LIN {X 0,Y 175.394,Z 402.692,A -85,B 0,C 180,E1 -25528.539,E2 -25528.539} C_VEL
LIN {X 0,Y 177.917,Z 390.914,A -85,B 0,C 180,E1 -25529.64,E2 -25529.64} C_VEL
LIN {X 0,Y 179.581,Z 378.992,A -85,B 0,C 180,E1 -25530.439,E2 -25530.439} C_VEL
LIN {X 0,Y 180.606,Z 365.157,A -85,B 0,C 180,E1 -25531.052,E2 -25531.052} C_VEL
LIN {X 0,Y 176.084,Z 356.031,A -85,B 0,C 180,E1 -25534.195,E2 -25534.195} C_VEL
LIN {X 0,Y 171.449,Z 347.762,A -85,B 0,C 180,E1 -25537.875,E2 -25537.875} C_VEL
LIN {X 0,Y 167.95,Z 342.316,A -85,B 0,C 180,E1 -25541.096,E2 -25541.096} C_VEL
LIN {X 0,Y 166.255,Z 339.586,A -85,B 0,C 180,E1 -25542.893,E2 -25542.893} C_VEL
LIN {X 0,Y 163.938,Z 336.007,A -85,B 0,C 180,E1 -25545.689,E2 -25545.689} C_VEL
LIN {X 0,Y 161.573,Z 332.428,A -85,B 0,C 180,E1 -25549.188,E2 -25549.188} C_VEL
LIN {X 0,Y 160.8,Z 331.442,A -85,B 0,C 180,E1 -25550.526,E2 -25550.526} C_VEL
LIN {X 0,Y 158.685,Z 328.085,A -85,B 0,C 180,E1 -25555.56,E2 -25555.56} C_VEL
LIN {X 0,Y 158.317,Z 327.018,A -85,B 0,C 180,E1 -25557.038,E2 -25557.038} C_VEL
LIN {X 0,Y 157.707,Z 326.481,A -85,B 0,C 180,E1 -25559.999,E2 -25559.999} C_VEL
LIN {X 0,Y 158.2,Z 327.003,A -85,B 0,C 180,E1 -25568.944,E2 -25568.944} C_VEL
LIN {X 0,Y 159.684,Z 330.432,A -85,B 0,C 180,E1 -25573.724,E2 -25573.724} C_VEL
LIN {X 0,Y 160.618,Z 331.804,A -85,B 0,C 180,E1 -25575.659,E2 -25575.659} C_VEL
LIN {X 0,Y 161.933,Z 334.433,A -85,B 0,C 180,E1 -25578.055,E2 -25578.055} C_VEL
LIN {X 0,Y 165.141,Z 341.155,A -85,B 0,C 180,E1 -25582.629,E2 -25582.629} C_VEL
LIN {X 0,Y 167.909,Z 347.295,A -85,B 0,C 180,E1 -25585.802,E2 -25585.802} C_VEL
LIN {X 0,Y 170.429,Z 353.215,A -85,B 0,C 180,E1 -25588.32,E2 -25588.32} C_VEL
LIN {X 0,Y 173.374,Z 360.584,A -85,B 0,C 180,E1 -25590.951,E2 -25590.951} C_VEL
LIN {X 0,Y 176.879,Z 370.457,A -85,B 0,C 180,E1 -25593.798,E2 -25593.798} C_VEL
LIN {X 0,Y 177.593,Z 373.058,A -85,B 0,C 180,E1 -25594.381,E2 -25594.381} C_VEL
LIN {X 0,Y 178.04,Z 394.466,A -85,B 0,C 180,E1 -25596.206,E2 -25596.206} C_VEL
LIN {X 0,Y 176.549,Z 407.501,A -85,B 0,C 180,E1 -25596.734,E2 -25596.734} C_VEL
LIN {X 0,Y 173.815,Z 420.614,A -85,B 0,C 180,E1 -25597.525,E2 -25597.525} C_VEL
LIN {X 0,Y 169.933,Z 433.758,A -85,B 0,C 180,E1 -25598.683,E2 -25598.683} C_VEL
LIN {X 0,Y 165.401,Z 445.411,A -85,B 0,C 180,E1 -25600.108,E2 -25600.108} C_VEL
LIN {X 0,Y 159.65,Z 457.154,A -85,B 0,C 180,E1 -25602.024,E2 -25602.024} C_VEL
LIN {X 0,Y 154.205,Z 466.649,A -85,B 0,C 180,E1 -25604.125,E2 -25604.125} C_VEL
LIN {X 0,Y 148.424,Z 475.35,A -85,B 0,C 180,E1 -25606.639,E2 -25606.639} C_VEL
LIN {X 0,Y 142.089,Z 483.85,A -85,B 0,C 180,E1 -25609.983,E2 -25609.983} C_VEL
LIN {X 0,Y 136.434,Z 490.753,A -85,B 0,C 180,E1 -25613.673,E2 -25613.673} C_VEL
LIN {X 0,Y 131.518,Z 496.334,A -85,B 0,C 180,E1 -25617.698,E2 -25617.698} C_VEL
LIN {X 0,Y 127.701,Z 500.475,A -85,B 0,C 180,E1 -25621.709,E2 -25621.709} C_VEL
LIN {X 0,Y 124.221,Z 504.173,A -85,B 0,C 180,E1 -25626.669,E2 -25626.669} C_VEL
LIN {X 0,Y 121.436,Z 507.281,A -85,B 0,C 180,E1 -25633.179,E2 -25633.179} C_VEL
LIN {X 0,Y 120.473,Z 508.774,A -85,B 0,C 180,E1 -25639.92,E2 -25639.92} C_VEL
LIN {X 0,Y 120.585,Z 508.949,A -85,B 0,C 180,E1 -25643.305,E2 -25643.305} C_VEL
LIN {X 0,Y 121.01,Z 508.736,A -85,B 0,C 180,E1 -25646.669,E2 -25646.669} C_VEL
LIN {X 0,Y 121.498,Z 508.07,A -85,B 0,C 180,E1 -25649.999,E2 -25649.999} C_VEL
LIN {X 0,Y 120.971,Z 506.799,A -85,B 0,C 180,E1 -25653.329,E2 -25653.329} C_VEL
LIN {X 0,Y 120.525,Z 504.589,A -85,B 0,C 180,E1 -25657.567,E2 -25657.567} C_VEL
LIN {X 0,Y 120.742,Z 500.25,A -85,B 0,C 180,E1 -25663.462,E2 -25663.462} C_VEL
LIN {X 0,Y 121.918,Z 495.31,A -85,B 0,C 180,E1 -25668.483,E2 -25668.483} C_VEL
LIN {X 0,Y 123.994,Z 489.089,A -85,B 0,C 180,E1 -25673.374,E2 -25673.374} C_VEL
LIN {X 0,Y 127.247,Z 481.256,A -85,B 0,C 180,E1 -25678.099,E2 -25678.099} C_VEL
LIN {X 0,Y 130.569,Z 473.197,A -85,B 0,C 180,E1 -25681.848,E2 -25681.848} C_VEL
LIN {X 0,Y 131.685,Z 468.98,A -85,B 0,C 180,E1 -25683.603,E2 -25683.603} C_VEL
LIN {X 0,Y 132.139,Z 461.767,A -85,B 0,C 180,E1 -25686.543,E2 -25686.543} C_VEL
LIN {X 0,Y 132.615,Z 454.126,A -85,B 0,C 180,E1 -25689.272,E2 -25689.272} C_VEL
LIN {X 0,Y 133.673,Z 449.2,A -85,B 0,C 180,E1 -25690.61,E2 -25690.61} C_VEL
LIN {X 0,Y 137.177,Z 438.275,A -85,B 0,C 180,E1 -25692.75,E2 -25692.75} C_VEL
LIN {X 0,Y 140.428,Z 426.165,A -85,B 0,C 180,E1 -25694.477,E2 -25694.477} C_VEL
LIN {X 0,Y 142.791,Z 413.232,A -85,B 0,C 180,E1 -25695.841,E2 -25695.841} C_VEL
LIN {X 0,Y 144.369,Z 400.263,A -85,B 0,C 180,E1 -25696.68,E2 -25696.68} C_VEL
LIN {X 0,Y 145.125,Z 387.045,A -85,B 0,C 180,E1 -25697.314,E2 -25697.314} C_VEL
LIN {X 0,Y 144.369,Z 355.275,A -85,B 0,C 180,E1 -25699.747,E2 -25699.747} C_VEL
LIN {X 0,Y 143.902,Z 344.092,A -85,B 0,C 180,E1 -25700.717,E2 -25700.717} C_VEL
LIN {X 0,Y 140.398,Z 334.16,A -85,B 0,C 180,E1 -25702.969,E2 -25702.969} C_VEL
LIN {X 0,Y 135.644,Z 322.943,A -85,B 0,C 180,E1 -25706.209,E2 -25706.209} C_VEL
LIN {X 0,Y 132.185,Z 316.035,A -85,B 0,C 180,E1 -25708.763,E2 -25708.763} C_VEL
LIN {X 0,Y 129.855,Z 311.656,A -85,B 0,C 180,E1 -25710.628,E2 -25710.628} C_VEL
LIN {X 0,Y 127.246,Z 306.989,A -85,B 0,C 180,E1 -25712.893,E2 -25712.893} C_VEL
LIN {X 0,Y 124.677,Z 303.799,A -85,B 0,C 180,E1 -25715.213,E2 -25715.213} C_VEL
LIN {X 0,Y 123.773,Z 302.321,A -85,B 0,C 180,E1 -25716.137,E2 -25716.137} C_VEL
LIN {X 0,Y 121.22,Z 299.89,A -85,B 0,C 180,E1 -25718.756,E2 -25718.756} C_VEL
LIN {X 0,Y 119.684,Z 297.038,A -85,B 0,C 180,E1 -25720.713,E2 -25720.713} C_VEL
LIN {X 0,Y 116.749,Z 294.976,A -85,B 0,C 180,E1 -25724.531,E2 -25724.531} C_VEL
LIN {X 0,Y 115.469,Z 292.543,A -85,B 0,C 180,E1 -25726.875,E2 -25726.875} C_VEL
LIN {X 0,Y 115.306,Z 291.427,A -85,B 0,C 180,E1 -25728.301,E2 -25728.301} C_VEL
LIN {X 0,Y 115.34,Z 291.094,A -85,B 0,C 180,E1 -25733.001,E2 -25733.001} C_VEL
LIN {X 0,Y 115.939,Z 291.002,A -85,B 0,C 180,E1 -25740.001,E2 -25740.001} C_VEL
LIN {X 0,Y 115.336,Z 291.08,A -85,B 0,C 180,E1 -25747.001,E2 -25747.001} C_VEL
LIN {X 0,Y 115.198,Z 291.126,A -85,B 0,C 180,E1 -25752.558,E2 -25752.558} C_VEL
LIN {X 0,Y 114.963,Z 291.274,A -85,B 0,C 180,E1 -25760.114,E2 -25760.114} C_VEL
LIN {X 0,Y 115.129,Z 292.227,A -85,B 0,C 180,E1 -25762.246,E2 -25762.246} C_VEL
LIN {X 0,Y 116.662,Z 295.146,A -85,B 0,C 180,E1 -25765.179,E2 -25765.179} C_VEL
LIN {X 0,Y 119.689,Z 297.275,A -85,B 0,C 180,E1 -25769.122,E2 -25769.122} C_VEL
LIN {X 0,Y 121.495,Z 300.418,A -85,B 0,C 180,E1 -25771.375,E2 -25771.375} C_VEL
LIN {X 0,Y 124.006,Z 302.79,A -85,B 0,C 180,E1 -25773.911,E2 -25773.911} C_VEL
LIN {X 0,Y 126.412,Z 306.25,A -85,B 0,C 180,E1 -25776.208,E2 -25776.208} C_VEL
LIN {X 0,Y 127.814,Z 307.903,A -85,B 0,C 180,E1 -25777.405,E2 -25777.405} C_VEL
LIN {X 0,Y 131.403,Z 312.946,A -85,B 0,C 180,E1 -25780.275,E2 -25780.275} C_VEL
LIN {X 0,Y 136.614,Z 320.749,A -85,B 0,C 180,E1 -25783.917,E2 -25783.917} C_VEL
LIN {X 0,Y 141.926,Z 329.84,A -85,B 0,C 180,E1 -25787.192,E2 -25787.192} C_VEL
LIN {X 0,Y 147.468,Z 341.166,A -85,B 0,C 180,E1 -25790.295,E2 -25790.295} C_VEL
LIN {X 0,Y 148.103,Z 342.665,A -85,B 0,C 180,E1 -25790.639,E2 -25790.639} C_VEL
LIN {X 0,Y 145.968,Z 378.464,A -85,B 0,C 180,E1 -25792.341,E2 -25792.341} C_VEL
LIN {X 0,Y 144.546,Z 391.684,A -85,B 0,C 180,E1 -25793.518,E2 -25793.518} C_VEL
LIN {X 0,Y 142.217,Z 404.62,A -85,B 0,C 180,E1 -25795.155,E2 -25795.155} C_VEL
LIN {X 0,Y 139.305,Z 416.238,A -85,B 0,C 180,E1 -25797.159,E2 -25797.159} C_VEL
LIN {X 0,Y 135.891,Z 427.426,A -85,B 0,C 180,E1 -25799.721,E2 -25799.721} C_VEL
LIN {X 0,Y 132.314,Z 437.523,A -85,B 0,C 180,E1 -25802.736,E2 -25802.736} C_VEL
LIN {X 0,Y 128.188,Z 447.433,A -85,B 0,C 180,E1 -25806.581,E2 -25806.581} C_VEL
LIN {X 0,Y 124.237,Z 456.159,A -85,B 0,C 180,E1 -25811.02,E2 -25811.02} C_VEL
LIN {X 0,Y 120.953,Z 463.158,A -85,B 0,C 180,E1 -25815.705,E2 -25815.705} C_VEL
LIN {X 0,Y 118.86,Z 467.887,A -85,B 0,C 180,E1 -25819.784,E2 -25819.784} C_VEL
LIN {X 0,Y 116.81,Z 472.507,A -85,B 0,C 180,E1 -25824.824,E2 -25824.824} C_VEL
LIN {X 0,Y 115.387,Z 476.063,A -85,B 0,C 180,E1 -25830.001,E2 -25830.001} C_VEL
LIN {X 0,Y 114.996,Z 477.866,A -85,B 0,C 180,E1 -25833.505,E2 -25833.505} C_VEL
LIN {X 0,Y 114.981,Z 479.23,A -85,B 0,C 180,E1 -25837.023,E2 -25837.023} C_VEL
LIN {X 0,Y 115.747,Z 480.843,A -85,B 0,C 180,E1 -25844.057,E2 -25844.057} C_VEL
LIN {X 0,Y 116.611,Z 481.045,A -85,B 0,C 180,E1 -25847.539,E2 -25847.539} C_VEL
LIN {X 0,Y 119.419,Z 480.261,A -85,B 0,C 180,E1 -25854.329,E2 -25854.329} C_VEL
LIN {X 0,Y 121.324,Z 479.292,A -85,B 0,C 180,E1 -25857.609,E2 -25857.609} C_VEL
LIN {X 0,Y 124.978,Z 476.922,A -85,B 0,C 180,E1 -25862.486,E2 -25862.486} C_VEL
LIN {X 0,Y 129.035,Z 473.733,A -85,B 0,C 180,E1 -25866.808,E2 -25866.808} C_VEL
LIN {X 0,Y 133.87,Z 469.359,A -85,B 0,C 180,E1 -25871.014,E2 -25871.014} C_VEL
LIN {X 0,Y 139.766,Z 463.195,A -85,B 0,C 180,E1 -25875.252,E2 -25875.252} C_VEL
LIN {X 0,Y 145.237,Z 456.626,A -85,B 0,C 180,E1 -25878.594,E2 -25878.594} C_VEL
LIN {X 0,Y 151.673,Z 447.723,A -85,B 0,C 180,E1 -25881.973,E2 -25881.973} C_VEL
LIN {X 0,Y 157.258,Z 438.48,A -85,B 0,C 180,E1 -25884.646,E2 -25884.646} C_VEL
LIN {X 0,Y 162.491,Z 428.091,A -85,B 0,C 180,E1 -25886.929,E2 -25886.929} C_VEL
LIN {X 0,Y 167.271,Z 416.474,A -85,B 0,C 180,E1 -25888.878,E2 -25888.878} C_VEL
LIN {X 0,Y 171.013,Z 404.942,A -85,B 0,C 180,E1 -25890.303,E2 -25890.303} C_VEL
LIN {X 0,Y 173.817,Z 392.872,A -85,B 0,C 180,E1 -25891.453,E2 -25891.453} C_VEL
LIN {X 0,Y 175.674,Z 380.377,A -85,B 0,C 180,E1 -25892.328,E2 -25892.328} C_VEL
LIN {X 0,Y 176.593,Z 368.296,A -85,B 0,C 180,E1 -25892.921,E2 -25892.921} C_VEL
LIN {X 0,Y 172.546,Z 359.917,A -85,B 0,C 180,E1 -25896.023,E2 -25896.023} C_VEL
LIN {X 0,Y 168.578,Z 352.796,A -85,B 0,C 180,E1 -25899.476,E2 -25899.476} C_VEL
LIN {X 0,Y 164.834,Z 346.457,A -85,B 0,C 180,E1 -25903.381,E2 -25903.381} C_VEL
LIN {X 0,Y 162.344,Z 342.538,A -85,B 0,C 180,E1 -25906.544,E2 -25906.544} C_VEL
LIN {X 0,Y 159.821,Z 338.501,A -85,B 0,C 180,E1 -25910.667,E2 -25910.667} C_VEL
LIN {X 0,Y 157.619,Z 334.901,A -85,B 0,C 180,E1 -25916.175,E2 -25916.175} C_VEL
LIN {X 0,Y 157.337,Z 333.996,A -85,B 0,C 180,E1 -25917.439,E2 -25917.439} C_VEL
LIN {X 0,Y 156.839,Z 333.527,A -85,B 0,C 180,E1 -25919.999,E2 -25919.999} C_VEL
LIN {X 0,Y 157.267,Z 334.047,A -85,B 0,C 180,E1 -25928.715,E2 -25928.715} C_VEL
LIN {X 0,Y 158.483,Z 337.194,A -85,B 0,C 180,E1 -25933.014,E2 -25933.014} C_VEL
LIN {X 0,Y 159.377,Z 338.564,A -85,B 0,C 180,E1 -25935.014,E2 -25935.014} C_VEL
LIN {X 0,Y 160.56,Z 341.163,A -85,B 0,C 180,E1 -25937.349,E2 -25937.349} C_VEL
LIN {X 0,Y 163.393,Z 347.576,A -85,B 0,C 180,E1 -25941.716,E2 -25941.716} C_VEL
LIN {X 0,Y 165.894,Z 353.546,A -85,B 0,C 180,E1 -25944.813,E2 -25944.813} C_VEL
LIN {X 0,Y 168.255,Z 359.473,A -85,B 0,C 180,E1 -25947.352,E2 -25947.352} C_VEL
LIN {X 0,Y 171.163,Z 367.368,A -85,B 0,C 180,E1 -25950.145,E2 -25950.145} C_VEL
LIN {X 0,Y 173.909,Z 375.764,A -85,B 0,C 180,E1 -25952.559,E2 -25952.559} C_VEL
LIN {X 0,Y 174.185,Z 395.482,A -85,B 0,C 180,E1 -25954.295,E2 -25954.295} C_VEL
LIN {X 0,Y 172.423,Z 408.632,A -85,B 0,C 180,E1 -25954.855,E2 -25954.855} C_VEL
LIN {X 0,Y 169.43,Z 421.797,A -85,B 0,C 180,E1 -25955.674,E2 -25955.674} C_VEL
LIN {X 0,Y 165.602,Z 433.914,A -85,B 0,C 180,E1 -25956.771,E2 -25956.771} C_VEL
LIN {X 0,Y 160.927,Z 445.315,A -85,B 0,C 180,E1 -25958.178,E2 -25958.178} C_VEL
LIN {X 0,Y 154.992,Z 456.921,A -85,B 0,C 180,E1 -25960.076,E2 -25960.076} C_VEL
LIN {X 0,Y 149.344,Z 466.307,A -85,B 0,C 180,E1 -25962.167,E2 -25962.167} C_VEL
LIN {X 0,Y 143.334,Z 474.897,A -85,B 0,C 180,E1 -25964.686,E2 -25964.686} C_VEL
LIN {X 0,Y 136.715,Z 483.315,A -85,B 0,C 180,E1 -25968.065,E2 -25968.065} C_VEL
LIN {X 0,Y 130.759,Z 490.158,A -85,B 0,C 180,E1 -25971.822,E2 -25971.822} C_VEL
LIN {X 0,Y 125.548,Z 495.687,A -85,B 0,C 180,E1 -25975.958,E2 -25975.958} C_VEL
LIN {X 0,Y 121.116,Z 500.11,A -85,B 0,C 180,E1 -25980.505,E2 -25980.505} C_VEL
LIN {X 0,Y 117.678,Z 503.427,A -85,B 0,C 180,E1 -25985.287,E2 -25985.287} C_VEL
LIN {X 0,Y 114.615,Z 506.482,A -85,B 0,C 180,E1 -25992.145,E2 -25992.145} C_VEL
LIN {X 0,Y 113.435,Z 507.922,A -85,B 0,C 180,E1 -25999.287,E2 -25999.287} C_VEL
LIN {X 0,Y 113.514,Z 508.08,A -85,B 0,C 180,E1 -26002.886,E2 -26002.886} C_VEL
LIN {X 0,Y 113.92,Z 507.847,A -85,B 0,C 180,E1 -26006.462,E2 -26006.462} C_VEL
LIN {X 0,Y 114.414,Z 507.144,A -85,B 0,C 180,E1 -26009.999,E2 -26009.999} C_VEL
LIN {X 0,Y 113.849,Z 505.845,A -85,B 0,C 180,E1 -26013.538,E2 -26013.538} C_VEL
LIN {X 0,Y 113.446,Z 503.845,A -85,B 0,C 180,E1 -26017.609,E2 -26017.609} C_VEL
LIN {X 0,Y 113.546,Z 500.609,A -85,B 0,C 180,E1 -26022.51,E2 -26022.51} C_VEL
LIN {X 0,Y 114.563,Z 496.012,A -85,B 0,C 180,E1 -26027.86,E2 -26027.86} C_VEL
LIN {X 0,Y 116.543,Z 490.195,A -85,B 0,C 180,E1 -26033.075,E2 -26033.075} C_VEL
LIN {X 0,Y 119.636,Z 482.958,A -85,B 0,C 180,E1 -26038.029,E2 -26038.029} C_VEL
LIN {X 0,Y 123.652,Z 473.951,A -85,B 0,C 180,E1 -26042.678,E2 -26042.678} C_VEL
LIN {X 0,Y 127.601,Z 464.73,A -85,B 0,C 180,E1 -26046.303,E2 -26046.303} C_VEL
LIN {X 0,Y 131.661,Z 454.571,A -85,B 0,C 180,E1 -26049.334,E2 -26049.334} C_VEL
LIN {X 0,Y 133.673,Z 449.2,A -85,B 0,C 180,E1 -26050.61,E2 -26050.61} C_VEL
LIN {X 0,Y 134.205,Z 445.842,A -85,B 0,C 180,E1 -26051.513,E2 -26051.513} C_VEL
LIN {X 0,Y 133.04,Z 434.995,A -85,B 0,C 180,E1 -26054.916,E2 -26054.916} C_VEL
LIN {X 0,Y 133.558,Z 431.399,A -85,B 0,C 180,E1 -26055.624,E2 -26055.624} C_VEL
LIN {X 0,Y 136.531,Z 418.477,A -85,B 0,C 180,E1 -26057.252,E2 -26057.252} C_VEL
LIN {X 0,Y 138.566,Z 405.274,A -85,B 0,C 180,E1 -26058.36,E2 -26058.36} C_VEL
LIN {X 0,Y 139.968,Z 388.759,A -85,B 0,C 180,E1 -26059.174,E2 -26059.174} C_VEL
LIN {X 0,Y 139.411,Z 356.425,A -85,B 0,C 180,E1 -26061.748,E2 -26061.748} C_VEL
LIN {X 0,Y 139.041,Z 346.487,A -85,B 0,C 180,E1 -26062.66,E2 -26062.66} C_VEL
LIN {X 0,Y 135.304,Z 335.775,A -85,B 0,C 180,E1 -26065.325,E2 -26065.325} C_VEL
LIN {X 0,Y 131.137,Z 325.959,A -85,B 0,C 180,E1 -26068.484,E2 -26068.484} C_VEL
LIN {X 0,Y 127.415,Z 318.054,A -85,B 0,C 180,E1 -26071.63,E2 -26071.63} C_VEL
LIN {X 0,Y 124.562,Z 312.954,A -85,B 0,C 180,E1 -26074.267,E2 -26074.267} C_VEL
LIN {X 0,Y 121.848,Z 309.113,A -85,B 0,C 180,E1 -26076.987,E2 -26076.987} C_VEL
LIN {X 0,Y 118.776,Z 305.609,A -85,B 0,C 180,E1 -26080.447,E2 -26080.447} C_VEL
LIN {X 0,Y 117.66,Z 303.597,A -85,B 0,C 180,E1 -26081.988,E2 -26081.988} C_VEL
LIN {X 0,Y 114.866,Z 301.207,A -85,B 0,C 180,E1 -26086.023,E2 -26086.023} C_VEL
LIN {X 0,Y 113.428,Z 298.165,A -85,B 0,C 180,E1 -26088.968,E2 -26088.968} C_VEL
LIN {X 0,Y 110.17,Z 295.549,A -85,B 0,C 180,E1 -26098.173,E2 -26098.173} C_VEL
LIN {X 0,Y 109.911,Z 294.776,A -85,B 0,C 180,E1 -26100.001,E2 -26100.001} C_VEL
LIN {X 0,Y 109.728,Z 295.533,A -85,B 0,C 180,E1 -26109.215,E2 -26109.215} C_VEL
LIN {X 0,Y 113.304,Z 298.397,A -85,B 0,C 180,E1 -26120.659,E2 -26120.659} C_VEL
LIN {X 0,Y 115.139,Z 301.842,A -85,B 0,C 180,E1 -26124.288,E2 -26124.288} C_VEL
LIN {X 0,Y 117.801,Z 303.938,A -85,B 0,C 180,E1 -26128.024,E2 -26128.024} C_VEL
LIN {X 0,Y 119.672,Z 307.023,A -85,B 0,C 180,E1 -26130.475,E2 -26130.475} C_VEL
LIN {X 0,Y 121.796,Z 309.262,A -85,B 0,C 180,E1 -26132.781,E2 -26132.781} C_VEL
LIN {X 0,Y 124.307,Z 312.734,A -85,B 0,C 180,E1 -26135.302,E2 -26135.302} C_VEL
LIN {X 0,Y 128.508,Z 318.707,A -85,B 0,C 180,E1 -26138.972,E2 -26138.972} C_VEL
LIN {X 0,Y 134.007,Z 327.357,A -85,B 0,C 180,E1 -26143.079,E2 -26143.079} C_VEL
LIN {X 0,Y 138.675,Z 335.928,A -85,B 0,C 180,E1 -26146.156,E2 -26146.156} C_VEL
LIN {X 0,Y 142.975,Z 345.095,A -85,B 0,C 180,E1 -26148.758,E2 -26148.758} C_VEL
LIN {X 0,Y 140.768,Z 379.531,A -85,B 0,C 180,E1 -26150.434,E2 -26150.434} C_VEL
LIN {X 0,Y 139.231,Z 392.988,A -85,B 0,C 180,E1 -26151.68,E2 -26151.68} C_VEL
LIN {X 0,Y 136.762,Z 405.663,A -85,B 0,C 180,E1 -26153.319,E2 -26153.319} C_VEL
LIN {X 0,Y 133.482,Z 418.016,A -85,B 0,C 180,E1 -26155.53,E2 -26155.53} C_VEL
LIN {X 0,Y 129.898,Z 429.033,A -85,B 0,C 180,E1 -26158.165,E2 -26158.165} C_VEL
LIN {X 0,Y 126.53,Z 437.955,A -85,B 0,C 180,E1 -26160.924,E2 -26160.924} C_VEL
LIN {X 0,Y 122.517,Z 447.156,A -85,B 0,C 180,E1 -26164.52,E2 -26164.52} C_VEL
LIN {X 0,Y 118.273,Z 456.065,A -85,B 0,C 180,E1 -26169.115,E2 -26169.115} C_VEL
LIN {X 0,Y 114.683,Z 463.256,A -85,B 0,C 180,E1 -26173.994,E2 -26173.994} C_VEL
LIN {X 0,Y 111.929,Z 469.004,A -85,B 0,C 180,E1 -26179.144,E2 -26179.144} C_VEL
LIN {X 0,Y 109.781,Z 473.565,A -85,B 0,C 180,E1 -26184.491,E2 -26184.491} C_VEL
LIN {X 0,Y 108.31,Z 477.072,A -85,B 0,C 180,E1 -26190.002,E2 -26190.002} C_VEL
LIN {X 0,Y 107.935,Z 478.825,A -85,B 0,C 180,E1 -26193.735,E2 -26193.735} C_VEL
LIN {X 0,Y 107.94,Z 480.168,A -85,B 0,C 180,E1 -26197.484,E2 -26197.484} C_VEL
LIN {X 0,Y 108.869,Z 481.726,A -85,B 0,C 180,E1 -26204.966,E2 -26204.966} C_VEL
LIN {X 0,Y 111.21,Z 481.665,A -85,B 0,C 180,E1 -26212.284,E2 -26212.284} C_VEL
LIN {X 0,Y 112.946,Z 481.06,A -85,B 0,C 180,E1 -26215.823,E2 -26215.823} C_VEL
LIN {X 0,Y 115.04,Z 480.055,A -85,B 0,C 180,E1 -26219.258,E2 -26219.258} C_VEL
LIN {X 0,Y 118.782,Z 477.79,A -85,B 0,C 180,E1 -26224.069,E2 -26224.069} C_VEL
LIN {X 0,Y 123.4,Z 474.404,A -85,B 0,C 180,E1 -26228.792,E2 -26228.792} C_VEL
LIN {X 0,Y 128.565,Z 469.969,A -85,B 0,C 180,E1 -26233.103,E2 -26233.103} C_VEL
LIN {X 0,Y 134.532,Z 464.045,A -85,B 0,C 180,E1 -26237.224,E2 -26237.224} C_VEL
LIN {X 0,Y 140.612,Z 457.081,A -85,B 0,C 180,E1 -26240.78,E2 -26240.78} C_VEL
LIN {X 0,Y 147.365,Z 448.096,A -85,B 0,C 180,E1 -26244.169,E2 -26244.169} C_VEL
LIN {X 0,Y 153.2,Z 438.697,A -85,B 0,C 180,E1 -26246.847,E2 -26246.847} C_VEL
LIN {X 0,Y 158.7,Z 428.176,A -85,B 0,C 180,E1 -26249.095,E2 -26249.095} C_VEL
LIN {X 0,Y 163.04,Z 417.974,A -85,B 0,C 180,E1 -26250.797,E2 -26250.797} C_VEL
LIN {X 0,Y 167.183,Z 405.779,A -85,B 0,C 180,E1 -26252.31,E2 -26252.31} C_VEL
LIN {X 0,Y 170.143,Z 393.56,A -85,B 0,C 180,E1 -26253.457,E2 -26253.457} C_VEL
LIN {X 0,Y 172.05,Z 381.25,A -85,B 0,C 180,E1 -26254.318,E2 -26254.318} C_VEL
LIN {X 0,Y 172.922,Z 371.794,A -85,B 0,C 180,E1 -26254.757,E2 -26254.757} C_VEL
LIN {X 0,Y 169.519,Z 364.677,A -85,B 0,C 180,E1 -26257.61,E2 -26257.61} C_VEL
LIN {X 0,Y 166.287,Z 358.582,A -85,B 0,C 180,E1 -26260.679,E2 -26260.679} C_VEL
LIN {X 0,Y 163.063,Z 352.834,A -85,B 0,C 180,E1 -26264.306,E2 -26264.306} C_VEL
LIN {X 0,Y 160.818,Z 349.072,A -85,B 0,C 180,E1 -26267.378,E2 -26267.378} C_VEL
LIN {X 0,Y 158.534,Z 345.243,A -85,B 0,C 180,E1 -26271.395,E2 -26271.395} C_VEL
LIN {X 0,Y 156.574,Z 341.704,A -85,B 0,C 180,E1 -26276.794,E2 -26276.794} C_VEL
LIN {X 0,Y 156.317,Z 340.91,A -85,B 0,C 180,E1 -26278.067,E2 -26278.067} C_VEL
LIN {X 0,Y 155.733,Z 340.575,A -85,B 0,C 180,E1 -26282.586,E2 -26282.586} C_VEL
LIN {X 0,Y 156.325,Z 341.176,A -85,B 0,C 180,E1 -26288.48,E2 -26288.48} C_VEL
LIN {X 0,Y 157.401,Z 344.087,A -85,B 0,C 180,E1 -26292.539,E2 -26292.539} C_VEL
LIN {X 0,Y 158.217,Z 345.5,A -85,B 0,C 180,E1 -26294.506,E2 -26294.506} C_VEL
LIN {X 0,Y 159.242,Z 347.974,A -85,B 0,C 180,E1 -26296.691,E2 -26296.691} C_VEL
LIN {X 0,Y 161.617,Z 353.809,A -85,B 0,C 180,E1 -26300.678,E2 -26300.678} C_VEL
LIN {X 0,Y 163.809,Z 359.449,A -85,B 0,C 180,E1 -26303.646,E2 -26303.646} C_VEL
LIN {X 0,Y 166.403,Z 366.39,A -85,B 0,C 180,E1 -26306.646,E2 -26306.646} C_VEL
LIN {X 0,Y 169.805,Z 376.804,A -85,B 0,C 180,E1 -26310.111,E2 -26310.111} C_VEL
LIN {X 0,Y 170.492,Z 379.624,A -85,B 0,C 180,E1 -26310.811,E2 -26310.811} C_VEL
LIN {X 0,Y 170.479,Z 396.668,A -85,B 0,C 180,E1 -26312.314,E2 -26312.314} C_VEL
LIN {X 0,Y 168.475,Z 409.773,A -85,B 0,C 180,E1 -26312.88,E2 -26312.88} C_VEL
LIN {X 0,Y 165.538,Z 421.84,A -85,B 0,C 180,E1 -26313.647,E2 -26313.647} C_VEL
LIN {X 0,Y 161.465,Z 434.012,A -85,B 0,C 180,E1 -26314.759,E2 -26314.759} C_VEL
LIN {X 0,Y 155.968,Z 446.66,A -85,B 0,C 180,E1 -26316.346,E2 -26316.346} C_VEL
LIN {X 0,Y 149.856,Z 457.799,A -85,B 0,C 180,E1 -26318.229,E2 -26318.229} C_VEL
LIN {X 0,Y 143.408,Z 467.753,A -85,B 0,C 180,E1 -26320.57,E2 -26320.57} C_VEL
LIN {X 0,Y 136.057,Z 477.445,A -85,B 0,C 180,E1 -26323.683,E2 -26323.683} C_VEL
LIN {X 0,Y 129.342,Z 485.214,A -85,B 0,C 180,E1 -26327.218,E2 -26327.218} C_VEL
LIN {X 0,Y 123.288,Z 491.52,A -85,B 0,C 180,E1 -26331.166,E2 -26331.166} C_VEL
LIN {X 0,Y 118.041,Z 496.596,A -85,B 0,C 180,E1 -26335.554,E2 -26335.554} C_VEL
LIN {X 0,Y 113.628,Z 500.58,A -85,B 0,C 180,E1 -26340.342,E2 -26340.342} C_VEL
LIN {X 0,Y 109.308,Z 504.393,A -85,B 0,C 180,E1 -26347.307,E2 -26347.307} C_VEL
LIN {X 0,Y 106.863,Z 506.557,A -85,B 0,C 180,E1 -26354.747,E2 -26354.747} C_VEL
LIN {X 0,Y 106.46,Z 507.214,A -85,B 0,C 180,E1 -26362.412,E2 -26362.412} C_VEL
LIN {X 0,Y 106.832,Z 506.949,A -85,B 0,C 180,E1 -26366.227,E2 -26366.227} C_VEL
LIN {X 0,Y 107.313,Z 506.216,A -85,B 0,C 180,E1 -26369.998,E2 -26369.998} C_VEL
LIN {X 0,Y 106.726,Z 504.89,A -85,B 0,C 180,E1 -26373.774,E2 -26373.774} C_VEL
LIN {X 0,Y 106.35,Z 502.052,A -85,B 0,C 180,E1 -26379.506,E2 -26379.506} C_VEL
LIN {X 0,Y 106.842,Z 498.146,A -85,B 0,C 180,E1 -26385.253,E2 -26385.253} C_VEL
LIN {X 0,Y 108.364,Z 493.098,A -85,B 0,C 180,E1 -26390.896,E2 -26390.896} C_VEL
LIN {X 0,Y 111.023,Z 486.781,A -85,B 0,C 180,E1 -26396.301,E2 -26396.301} C_VEL
LIN {X 0,Y 114.582,Z 479.246,A -85,B 0,C 180,E1 -26401.215,E2 -26401.215} C_VEL
LIN {X 0,Y 118.449,Z 470.947,A -85,B 0,C 180,E1 -26405.343,E2 -26405.343} C_VEL
LIN {X 0,Y 122.822,Z 461.204,A -85,B 0,C 180,E1 -26409.005,E2 -26409.005} C_VEL
LIN {X 0,Y 126.767,Z 451.736,A -85,B 0,C 180,E1 -26411.701,E2 -26411.701} C_VEL
LIN {X 0,Y 130.997,Z 440.017,A -85,B 0,C 180,E1 -26414.22,E2 -26414.22} C_VEL
LIN {X 0,Y 133.558,Z 431.399,A -85,B 0,C 180,E1 -26415.624,E2 -26415.624} C_VEL
LIN {X 0,Y 134.488,Z 425.978,A -85,B 0,C 180,E1 -26416.538,E2 -26416.538} C_VEL
LIN {X 0,Y 134.201,Z 417.05,A -85,B 0,C 180,E1 -26418.383,E2 -26418.383} C_VEL
LIN {X 0,Y 133.61,Z 407.919,A -85,B 0,C 180,E1 -26420.045,E2 -26420.045} C_VEL
LIN {X 0,Y 133.887,Z 402.174,A -85,B 0,C 180,E1 -26420.634,E2 -26420.634} C_VEL
LIN {X 0,Y 134.953,Z 388.522,A -85,B 0,C 180,E1 -26421.324,E2 -26421.324} C_VEL
LIN {X 0,Y 134.652,Z 358.247,A -85,B 0,C 180,E1 -26423.83,E2 -26423.83} C_VEL
LIN {X 0,Y 134.437,Z 349.164,A -85,B 0,C 180,E1 -26424.672,E2 -26424.672} C_VEL
LIN {X 0,Y 131.156,Z 339.497,A -85,B 0,C 180,E1 -26427.257,E2 -26427.257} C_VEL
LIN {X 0,Y 127.084,Z 329.343,A -85,B 0,C 180,E1 -26430.721,E2 -26430.721} C_VEL
LIN {X 0,Y 123.722,Z 322.276,A -85,B 0,C 180,E1 -26433.882,E2 -26433.882} C_VEL
LIN {X 0,Y 121.817,Z 318.702,A -85,B 0,C 180,E1 -26435.842,E2 -26435.842} C_VEL
LIN {X 0,Y 119.112,Z 314.832,A -85,B 0,C 180,E1 -26438.815,E2 -26438.815} C_VEL
LIN {X 0,Y 116.583,Z 311.568,A -85,B 0,C 180,E1 -26442.002,E2 -26442.002} C_VEL
LIN {X 0,Y 115.825,Z 310.206,A -85,B 0,C 180,E1 -26443.136,E2 -26443.136} C_VEL
LIN {X 0,Y 113.192,Z 307.611,A -85,B 0,C 180,E1 -26447.317,E2 -26447.317} C_VEL
LIN {X 0,Y 111.979,Z 304.899,A -85,B 0,C 180,E1 -26450.062,E2 -26450.062} C_VEL
LIN {X 0,Y 109.205,Z 302.558,A -85,B 0,C 180,E1 -26458.618,E2 -26458.618} C_VEL
LIN {X 0,Y 109.016,Z 302.014,A -85,B 0,C 180,E1 -26460.001,E2 -26460.001} C_VEL
LIN {X 0,Y 108.764,Z 302.447,A -85,B 0,C 180,E1 -26468.361,E2 -26468.361} C_VEL
LIN {X 0,Y 111.939,Z 305.155,A -85,B 0,C 180,E1 -26479.721,E2 -26479.721} C_VEL
LIN {X 0,Y 113.421,Z 308.253,A -85,B 0,C 180,E1 -26482.974,E2 -26482.974} C_VEL
LIN {X 0,Y 115.955,Z 310.588,A -85,B 0,C 180,E1 -26486.885,E2 -26486.885} C_VEL
LIN {X 0,Y 118.257,Z 314.032,A -85,B 0,C 180,E1 -26490.004,E2 -26490.004} C_VEL
LIN {X 0,Y 119.602,Z 315.575,A -85,B 0,C 180,E1 -26491.558,E2 -26491.558} C_VEL
LIN {X 0,Y 122.983,Z 320.467,A -85,B 0,C 180,E1 -26495.125,E2 -26495.125} C_VEL
LIN {X 0,Y 125.862,Z 324.785,A -85,B 0,C 180,E1 -26497.771,E2 -26497.771} C_VEL
LIN {X 0,Y 130.974,Z 333.201,A -85,B 0,C 180,E1 -26501.875,E2 -26501.875} C_VEL
LIN {X 0,Y 135.145,Z 341.396,A -85,B 0,C 180,E1 -26504.855,E2 -26504.855} C_VEL
LIN {X 0,Y 137.996,Z 347.5,A -85,B 0,C 180,E1 -26506.73,E2 -26506.73} C_VEL
LIN {X 0,Y 135.777,Z 380.332,A -85,B 0,C 180,E1 -26508.372,E2 -26508.372} C_VEL
LIN {X 0,Y 134.198,Z 393.29,A -85,B 0,C 180,E1 -26509.578,E2 -26509.578} C_VEL
LIN {X 0,Y 131.734,Z 405.686,A -85,B 0,C 180,E1 -26511.184,E2 -26511.184} C_VEL
LIN {X 0,Y 128.754,Z 416.668,A -85,B 0,C 180,E1 -26513.102,E2 -26513.102} C_VEL
LIN {X 0,Y 124.925,Z 428.089,A -85,B 0,C 180,E1 -26515.768,E2 -26515.768} C_VEL
LIN {X 0,Y 120.881,Z 438.372,A -85,B 0,C 180,E1 -26518.939,E2 -26518.939} C_VEL
LIN {X 0,Y 117.02,Z 446.814,A -85,B 0,C 180,E1 -26522.263,E2 -26522.263} C_VEL
LIN {X 0,Y 113.2,Z 454.59,A -85,B 0,C 180,E1 -26526.202,E2 -26526.202} C_VEL
LIN {X 0,Y 109.15,Z 462.212,A -85,B 0,C 180,E1 -26531.222,E2 -26531.222} C_VEL
LIN {X 0,Y 105.929,Z 468.323,A -85,B 0,C 180,E1 -26536.575,E2 -26536.575} C_VEL
LIN {X 0,Y 103.425,Z 473.203,A -85,B 0,C 180,E1 -26542.191,E2 -26542.191} C_VEL
LIN {X 0,Y 101.63,Z 477.005,A -85,B 0,C 180,E1 -26548.02,E2 -26548.02} C_VEL
LIN {X 0,Y 100.876,Z 479.783,A -85,B 0,C 180,E1 -26553.997,E2 -26553.997} C_VEL
LIN {X 0,Y 100.908,Z 481.104,A -85,B 0,C 180,E1 -26558.009,E2 -26558.009} C_VEL
LIN {X 0,Y 101.713,Z 482.446,A -85,B 0,C 180,E1 -26564.677,E2 -26564.677} C_VEL
LIN {X 0,Y 103.105,Z 482.735,A -85,B 0,C 180,E1 -26569.928,E2 -26569.928} C_VEL
LIN {X 0,Y 106.566,Z 481.859,A -85,B 0,C 180,E1 -26577.495,E2 -26577.495} C_VEL
LIN {X 0,Y 108.867,Z 480.807,A -85,B 0,C 180,E1 -26581.095,E2 -26581.095} C_VEL
LIN {X 0,Y 112.674,Z 478.665,A -85,B 0,C 180,E1 -26585.817,E2 -26585.817} C_VEL
LIN {X 0,Y 117.903,Z 475.065,A -85,B 0,C 180,E1 -26590.973,E2 -26590.973} C_VEL
LIN {X 0,Y 123.422,Z 470.567,A -85,B 0,C 180,E1 -26595.381,E2 -26595.381} C_VEL
LIN {X 0,Y 130.623,Z 463.694,A -85,B 0,C 180,E1 -26600.059,E2 -26600.059} C_VEL
LIN {X 0,Y 137.353,Z 456.191,A -85,B 0,C 180,E1 -26603.696,E2 -26603.696} C_VEL
LIN {X 0,Y 144.164,Z 447.117,A -85,B 0,C 180,E1 -26606.917,E2 -26606.917} C_VEL
LIN {X 0,Y 150.03,Z 437.847,A -85,B 0,C 180,E1 -26609.401,E2 -26609.401} C_VEL
LIN {X 0,Y 155.135,Z 428.262,A -85,B 0,C 180,E1 -26611.37,E2 -26611.37} C_VEL
LIN {X 0,Y 159.664,Z 417.894,A -85,B 0,C 180,E1 -26613.038,E2 -26613.038} C_VEL
LIN {X 0,Y 163.618,Z 406.442,A -85,B 0,C 180,E1 -26614.425,E2 -26614.425} C_VEL
LIN {X 0,Y 166.695,Z 394.165,A -85,B 0,C 180,E1 -26615.559,E2 -26615.559} C_VEL
LIN {X 0,Y 168.712,Z 381.66,A -85,B 0,C 180,E1 -26616.412,E2 -26616.412} C_VEL
LIN {X 0,Y 169.312,Z 375.109,A -85,B 0,C 180,E1 -26616.769,E2 -26616.769} C_VEL
LIN {X 0,Y 165.86,Z 367.782,A -85,B 0,C 180,E1 -26620.029,E2 -26620.029} C_VEL
LIN {X 0,Y 162.878,Z 362.161,A -85,B 0,C 180,E1 -26623.283,E2 -26623.283} C_VEL
LIN {X 0,Y 160.884,Z 358.443,A -85,B 0,C 180,E1 -26625.866,E2 -26625.866} C_VEL
LIN {X 0,Y 159.299,Z 355.6,A -85,B 0,C 180,E1 -26628.266,E2 -26628.266} C_VEL
LIN {X 0,Y 157.425,Z 352.157,A -85,B 0,C 180,E1 -26631.818,E2 -26631.818} C_VEL
LIN {X 0,Y 155.548,Z 348.533,A -85,B 0,C 180,E1 -26637.41,E2 -26637.41} C_VEL
LIN {X 0,Y 155.315,Z 347.829,A -85,B 0,C 180,E1 -26638.703,E2 -26638.703} C_VEL
LIN {X 0,Y 154.852,Z 347.652,A -85,B 0,C 180,E1 -26643.17,E2 -26643.17} C_VEL
LIN {X 0,Y 155.347,Z 348.114,A -85,B 0,C 180,E1 -26647.983,E2 -26647.983} C_VEL
LIN {X 0,Y 156.535,Z 351.286,A -85,B 0,C 180,E1 -26652.61,E2 -26652.61} C_VEL
LIN {X 0,Y 157.544,Z 353.596,A -85,B 0,C 180,E1 -26655.11,E2 -26655.11} C_VEL
LIN {X 0,Y 159.799,Z 359.758,A -85,B 0,C 180,E1 -26659.458,E2 -26659.458} C_VEL
LIN {X 0,Y 161.839,Z 365.503,A -85,B 0,C 180,E1 -26662.514,E2 -26662.514} C_VEL
LIN {X 0,Y 164.361,Z 372.915,A -85,B 0,C 180,E1 -26665.702,E2 -26665.702} C_VEL
LIN {X 0,Y 167.163,Z 382.386,A -85,B 0,C 180,E1 -26668.832,E2 -26668.832} C_VEL
LIN {X 0,Y 167.042,Z 397.186,A -85,B 0,C 180,E1 -26670.212,E2 -26670.212} C_VEL
LIN {X 0,Y 164.864,Z 410.268,A -85,B 0,C 180,E1 -26670.786,E2 -26670.786} C_VEL
LIN {X 0,Y 161.285,Z 423.496,A -85,B 0,C 180,E1 -26671.637,E2 -26671.637} C_VEL
LIN {X 0,Y 156.793,Z 435.879,A -85,B 0,C 180,E1 -26672.813,E2 -26672.813} C_VEL
LIN {X 0,Y 151.878,Z 446.57,A -85,B 0,C 180,E1 -26674.193,E2 -26674.193} C_VEL
LIN {X 0,Y 145.576,Z 457.52,A -85,B 0,C 180,E1 -26676.036,E2 -26676.036} C_VEL
LIN {X 0,Y 138.883,Z 467.375,A -85,B 0,C 180,E1 -26678.338,E2 -26678.338} C_VEL
LIN {X 0,Y 132.474,Z 475.489,A -85,B 0,C 180,E1 -26680.887,E2 -26680.887} C_VEL
LIN {X 0,Y 125.343,Z 483.508,A -85,B 0,C 180,E1 -26684.365,E2 -26684.365} C_VEL
LIN {X 0,Y 119.883,Z 488.981,A -85,B 0,C 180,E1 -26687.609,E2 -26687.609} C_VEL
LIN {X 0,Y 113.981,Z 494.396,A -85,B 0,C 180,E1 -26691.931,E2 -26691.931} C_VEL
LIN {X 0,Y 108.114,Z 499.35,A -85,B 0,C 180,E1 -26697.678,E2 -26697.678} C_VEL
LIN {X 0,Y 104.855,Z 501.941,A -85,B 0,C 180,E1 -26702.018,E2 -26702.018} C_VEL
LIN {X 0,Y 102.732,Z 503.621,A -85,B 0,C 180,E1 -26705.765,E2 -26705.765} C_VEL
LIN {X 0,Y 99.97,Z 505.726,A -85,B 0,C 180,E1 -26713.667,E2 -26713.667} C_VEL
LIN {X 0,Y 99.39,Z 506.344,A -85,B 0,C 180,E1 -26721.868,E2 -26721.868} C_VEL
LIN {X 0,Y 99.749,Z 506.043,A -85,B 0,C 180,E1 -26725.958,E2 -26725.958} C_VEL
LIN {X 0,Y 100.211,Z 505.287,A -85,B 0,C 180,E1 -26729.998,E2 -26729.998} C_VEL
LIN {X 0,Y 99.599,Z 503.935,A -85,B 0,C 180,E1 -26734.045,E2 -26734.045} C_VEL
LIN {X 0,Y 99.282,Z 501.047,A -85,B 0,C 180,E1 -26740.191,E2 -26740.191} C_VEL
LIN {X 0,Y 99.941,Z 497.095,A -85,B 0,C 180,E1 -26746.335,E2 -26746.335} C_VEL
LIN {X 0,Y 101.681,Z 491.994,A -85,B 0,C 180,E1 -26752.341,E2 -26752.341} C_VEL
LIN {X 0,Y 104.66,Z 485.627,A -85,B 0,C 180,E1 -26758.035,E2 -26758.035} C_VEL
LIN {X 0,Y 108.689,Z 477.709,A -85,B 0,C 180,E1 -26763.339,E2 -26763.339} C_VEL
LIN {X 0,Y 113.535,Z 467.79,A -85,B 0,C 180,E1 -26768.241,E2 -26768.241} C_VEL
LIN {X 0,Y 117.925,Z 458.709,A -85,B 0,C 180,E1 -26771.527,E2 -26771.527} C_VEL
LIN {X 0,Y 122.564,Z 447.458,A -85,B 0,C 180,E1 -26774.619,E2 -26774.619} C_VEL
LIN {X 0,Y 125.93,Z 438.244,A -85,B 0,C 180,E1 -26776.508,E2 -26776.508} C_VEL
LIN {X 0,Y 129.731,Z 425.447,A -85,B 0,C 180,E1 -26778.438,E2 -26778.438} C_VEL
LIN {X 0,Y 132.487,Z 412.018,A -85,B 0,C 180,E1 -26779.923,E2 -26779.923} C_VEL
LIN {X 0,Y 133.887,Z 402.174,A -85,B 0,C 180,E1 -26780.634,E2 -26780.634} C_VEL
LIN {X 0,Y 134.12,Z 398.324,A -85,B 0,C 180,E1 -26780.956,E2 -26780.956} C_VEL
LIN {X 0,Y 133.633,Z 392.686,A -85,B 0,C 180,E1 -26781.704,E2 -26781.704} C_VEL
LIN {X 0,Y 130.995,Z 379.921,A -85,B 0,C 180,E1 -26783.939,E2 -26783.939} C_VEL
LIN {X 0,Y 130.254,Z 374.257,A -85,B 0,C 180,E1 -26784.751,E2 -26784.751} C_VEL
LIN {X 0,Y 130.173,Z 372.312,A -85,B 0,C 180,E1 -26784.954,E2 -26784.954} C_VEL
LIN {X 0,Y 129.97,Z 351.733,A -85,B 0,C 180,E1 -26786.848,E2 -26786.848} C_VEL
LIN {X 0,Y 126.342,Z 340.863,A -85,B 0,C 180,E1 -26790.073,E2 -26790.073} C_VEL
LIN {X 0,Y 122.951,Z 332.318,A -85,B 0,C 180,E1 -26793.362,E2 -26793.362} C_VEL
LIN {X 0,Y 120.468,Z 326.891,A -85,B 0,C 180,E1 -26796.012,E2 -26796.012} C_VEL
LIN {X 0,Y 119.303,Z 324.601,A -85,B 0,C 180,E1 -26797.344,E2 -26797.344} C_VEL
LIN {X 0,Y 116.926,Z 321.05,A -85,B 0,C 180,E1 -26800.192,E2 -26800.192} C_VEL
LIN {X 0,Y 114.431,Z 317.404,A -85,B 0,C 180,E1 -26803.699,E2 -26803.699} C_VEL
LIN {X 0,Y 113.602,Z 316.437,A -85,B 0,C 180,E1 -26804.986,E2 -26804.986} C_VEL
LIN {X 0,Y 111.379,Z 313.644,A -85,B 0,C 180,E1 -26809.089,E2 -26809.089} C_VEL
LIN {X 0,Y 110.506,Z 311.676,A -85,B 0,C 180,E1 -26811.313,E2 -26811.313} C_VEL
LIN {X 0,Y 108.169,Z 309.336,A -85,B 0,C 180,E1 -26819.652,E2 -26819.652} C_VEL
LIN {X 0,Y 107.748,Z 309.172,A -85,B 0,C 180,E1 -26825.616,E2 -26825.616} C_VEL
LIN {X 0,Y 108.369,Z 310.251,A -85,B 0,C 180,E1 -26831.716,E2 -26831.716} C_VEL
LIN {X 0,Y 110.615,Z 312.136,A -85,B 0,C 180,E1 -26838.841,E2 -26838.841} C_VEL
LIN {X 0,Y 112.188,Z 315.244,A -85,B 0,C 180,E1 -26842.453,E2 -26842.453} C_VEL
LIN {X 0,Y 114.263,Z 317.33,A -85,B 0,C 180,E1 -26845.867,E2 -26845.867} C_VEL
LIN {X 0,Y 116.868,Z 321.058,A -85,B 0,C 180,E1 -26849.544,E2 -26849.544} C_VEL
LIN {X 0,Y 120.602,Z 326.626,A -85,B 0,C 180,E1 -26853.867,E2 -26853.867} C_VEL
LIN {X 0,Y 124.265,Z 332.489,A -85,B 0,C 180,E1 -26857.432,E2 -26857.432} C_VEL
LIN {X 0,Y 128.723,Z 340.487,A -85,B 0,C 180,E1 -26861.196,E2 -26861.196} C_VEL
LIN {X 0,Y 133.183,Z 350.107,A -85,B 0,C 180,E1 -26864.562,E2 -26864.562} C_VEL
LIN {X 0,Y 130.935,Z 381.452,A -85,B 0,C 180,E1 -26866.176,E2 -26866.176} C_VEL
LIN {X 0,Y 129.178,Z 394.803,A -85,B 0,C 180,E1 -26867.459,E2 -26867.459} C_VEL
LIN {X 0,Y 126.351,Z 407.724,A -85,B 0,C 180,E1 -26869.192,E2 -26869.192} C_VEL
LIN {X 0,Y 122.717,Z 419.996,A -85,B 0,C 180,E1 -26871.481,E2 -26871.481} C_VEL
LIN {X 0,Y 118.72,Z 430.958,A -85,B 0,C 180,E1 -26874.229,E2 -26874.229} C_VEL
LIN {X 0,Y 114.451,Z 440.834,A -85,B 0,C 180,E1 -26877.502,E2 -26877.502} C_VEL
LIN {X 0,Y 109.996,Z 449.802,A -85,B 0,C 180,E1 -26881.369,E2 -26881.369} C_VEL
LIN {X 0,Y 105.225,Z 458.557,A -85,B 0,C 180,E1 -26886.378,E2 -26886.378} C_VEL
LIN {X 0,Y 101.203,Z 465.592,A -85,B 0,C 180,E1 -26891.792,E2 -26891.792} C_VEL
LIN {X 0,Y 98.092,Z 471.193,A -85,B 0,C 180,E1 -26897.59,E2 -26897.59} C_VEL
LIN {X 0,Y 95.713,Z 475.641,A -85,B 0,C 180,E1 -26903.678,E2 -26903.678} C_VEL
LIN {X 0,Y 94.154,Z 479.053,A -85,B 0,C 180,E1 -26910.002,E2 -26910.002} C_VEL
LIN {X 0,Y 93.82,Z 480.74,A -85,B 0,C 180,E1 -26914.298,E2 -26914.298} C_VEL
LIN {X 0,Y 93.888,Z 482.04,A -85,B 0,C 180,E1 -26918.612,E2 -26918.612} C_VEL
LIN {X 0,Y 94.773,Z 483.292,A -85,B 0,C 180,E1 -26925.409,E2 -26925.409} C_VEL
LIN {X 0,Y 96.445,Z 483.579,A -85,B 0,C 180,E1 -26931.369,E2 -26931.369} C_VEL
LIN {X 0,Y 100.296,Z 482.654,A -85,B 0,C 180,E1 -26939.375,E2 -26939.375} C_VEL
LIN {X 0,Y 102.82,Z 481.557,A -85,B 0,C 180,E1 -26943.15,E2 -26943.15} C_VEL
LIN {X 0,Y 106.699,Z 479.532,A -85,B 0,C 180,E1 -26947.774,E2 -26947.774} C_VEL
LIN {X 0,Y 112.608,Z 475.713,A -85,B 0,C 180,E1 -26953.356,E2 -26953.356} C_VEL
LIN {X 0,Y 118.502,Z 471.158,A -85,B 0,C 180,E1 -26957.846,E2 -26957.846} C_VEL
LIN {X 0,Y 126.142,Z 464.222,A -85,B 0,C 180,E1 -26962.555,E2 -26962.555} C_VEL
LIN {X 0,Y 133.246,Z 456.621,A -85,B 0,C 180,E1 -26966.174,E2 -26966.174} C_VEL
LIN {X 0,Y 140.289,Z 447.572,A -85,B 0,C 180,E1 -26969.331,E2 -26969.331} C_VEL
LIN {X 0,Y 146.513,Z 438.068,A -85,B 0,C 180,E1 -26971.814,E2 -26971.814} C_VEL
LIN {X 0,Y 151.814,Z 428.345,A -85,B 0,C 180,E1 -26973.758,E2 -26973.758} C_VEL
LIN {X 0,Y 156.453,Z 417.959,A -85,B 0,C 180,E1 -26975.35,E2 -26975.35} C_VEL
LIN {X 0,Y 160.641,Z 405.939,A -85,B 0,C 180,E1 -26976.743,E2 -26976.743} C_VEL
LIN {X 0,Y 163.541,Z 394.458,A -85,B 0,C 180,E1 -26977.776,E2 -26977.776} C_VEL
LIN {X 0,Y 165.624,Z 381.892,A -85,B 0,C 180,E1 -26978.604,E2 -26978.604} C_VEL
LIN {X 0,Y 165.907,Z 378.699,A -85,B 0,C 180,E1 -26978.798,E2 -26978.798} C_VEL
LIN {X 0,Y 162.61,Z 371.457,A -85,B 0,C 180,E1 -26982.389,E2 -26982.389} C_VEL
LIN {X 0,Y 159.441,Z 365.176,A -85,B 0,C 180,E1 -26986.538,E2 -26986.538} C_VEL
LIN {X 0,Y 157.863,Z 362.208,A -85,B 0,C 180,E1 -26989.093,E2 -26989.093} C_VEL
LIN {X 0,Y 156.143,Z 358.858,A -85,B 0,C 180,E1 -26992.646,E2 -26992.646} C_VEL
LIN {X 0,Y 154.443,Z 354.905,A -85,B 0,C 180,E1 -26998.696,E2 -26998.696} C_VEL
LIN {X 0,Y 153.999,Z 354.65,A -85,B 0,C 180,E1 -27002.615,E2 -27002.615} C_VEL
LIN {X 0,Y 154.396,Z 355.096,A -85,B 0,C 180,E1 -27007.574,E2 -27007.574} C_VEL
LIN {X 0,Y 155.908,Z 359.173,A -85,B 0,C 180,E1 -27013.366,E2 -27013.366} C_VEL
LIN {X 0,Y 158.133,Z 365.957,A -85,B 0,C 180,E1 -27018.345,E2 -27018.345} C_VEL
LIN {X 0,Y 160.029,Z 371.774,A -85,B 0,C 180,E1 -27021.489,E2 -27021.489} C_VEL
LIN {X 0,Y 162.45,Z 379.772,A -85,B 0,C 180,E1 -27024.847,E2 -27024.847} C_VEL
LIN {X 0,Y 164.103,Z 386.008,A -85,B 0,C 180,E1 -27026.916,E2 -27026.916} C_VEL
LIN {X 0,Y 163.708,Z 398.704,A -85,B 0,C 180,E1 -27028.067,E2 -27028.067} C_VEL
LIN {X 0,Y 161.1,Z 412.185,A -85,B 0,C 180,E1 -27028.697,E2 -27028.697} C_VEL
LIN {X 0,Y 157.517,Z 424.377,A -85,B 0,C 180,E1 -27029.485,E2 -27029.485} C_VEL
LIN {X 0,Y 153.062,Z 435.965,A -85,B 0,C 180,E1 -27030.58,E2 -27030.58} C_VEL
LIN {X 0,Y 147.295,Z 447.732,A -85,B 0,C 180,E1 -27032.122,E2 -27032.122} C_VEL
LIN {X 0,Y 140.813,Z 458.317,A -85,B 0,C 180,E1 -27033.926,E2 -27033.926} C_VEL
LIN {X 0,Y 134.583,Z 466.998,A -85,B 0,C 180,E1 -27035.961,E2 -27035.961} C_VEL
LIN {X 0,Y 127.937,Z 475.033,A -85,B 0,C 180,E1 -27038.482,E2 -27038.482} C_VEL
LIN {X 0,Y 120.478,Z 482.959,A -85,B 0,C 180,E1 -27041.947,E2 -27041.947} C_VEL
LIN {X 0,Y 112.537,Z 490.289,A -85,B 0,C 180,E1 -27046.609,E2 -27046.609} C_VEL
LIN {X 0,Y 106.556,Z 495.258,A -85,B 0,C 180,E1 -27051.201,E2 -27051.201} C_VEL
LIN {X 0,Y 101.45,Z 499.144,A -85,B 0,C 180,E1 -27056.343,E2 -27056.343} C_VEL
LIN {X 0,Y 98.606,Z 501.202,A -85,B 0,C 180,E1 -27060.071,E2 -27060.071} C_VEL
LIN {X 0,Y 96.25,Z 502.842,A -85,B 0,C 180,E1 -27064.015,E2 -27064.015} C_VEL
LIN {X 0,Y 93.131,Z 504.897,A -85,B 0,C 180,E1 -27072.43,E2 -27072.43} C_VEL
LIN {X 0,Y 92.336,Z 505.469,A -85,B 0,C 180,E1 -27081.242,E2 -27081.242} C_VEL
LIN {X 0,Y 92.666,Z 505.135,A -85,B 0,C 180,E1 -27085.649,E2 -27085.649} C_VEL
LIN {X 0,Y 93.108,Z 504.358,A -85,B 0,C 180,E1 -27089.998,E2 -27089.998} C_VEL
LIN {X 0,Y 92.254,Z 501.511,A -85,B 0,C 180,E1 -27097.971,E2 -27097.971} C_VEL
LIN {X 0,Y 92.655,Z 497.519,A -85,B 0,C 180,E1 -27105.393,E2 -27105.393} C_VEL
LIN {X 0,Y 94.258,Z 492.757,A -85,B 0,C 180,E1 -27111.886,E2 -27111.886} C_VEL
LIN {X 0,Y 97.12,Z 486.748,A -85,B 0,C 180,E1 -27118.056,E2 -27118.056} C_VEL
LIN {X 0,Y 101.199,Z 479.293,A -85,B 0,C 180,E1 -27123.748,E2 -27123.748} C_VEL
LIN {X 0,Y 106.172,Z 470.054,A -85,B 0,C 180,E1 -27128.962,E2 -27128.962} C_VEL
LIN {X 0,Y 111.035,Z 460.502,A -85,B 0,C 180,E1 -27132.873,E2 -27132.873} C_VEL
LIN {X 0,Y 115.382,Z 451.241,A -85,B 0,C 180,E1 -27135.697,E2 -27135.697} C_VEL
LIN {X 0,Y 119.994,Z 439.787,A -85,B 0,C 180,E1 -27138.307,E2 -27138.307} C_VEL
LIN {X 0,Y 123.908,Z 427.879,A -85,B 0,C 180,E1 -27140.283,E2 -27140.283} C_VEL
LIN {X 0,Y 126.875,Z 415.157,A -85,B 0,C 180,E1 -27141.847,E2 -27141.847} C_VEL
LIN {X 0,Y 129.064,Z 401.765,A -85,B 0,C 180,E1 -27142.905,E2 -27142.905} C_VEL
LIN {X 0,Y 130.126,Z 389.367,A -85,B 0,C 180,E1 -27143.552,E2 -27143.552} C_VEL
LIN {X 0,Y 130.173,Z 372.312,A -85,B 0,C 180,E1 -27144.954,E2 -27144.954} C_VEL
LIN {X 0,Y 129.605,Z 367.335,A -85,B 0,C 180,E1 -27145.686,E2 -27145.686} C_VEL
LIN {X 0,Y 128.383,Z 362.767,A -85,B 0,C 180,E1 -27146.77,E2 -27146.77} C_VEL
LIN {X 0,Y 125.533,Z 353.946,A -85,B 0,C 180,E1 -27149.32,E2 -27149.32} C_VEL
LIN {X 0,Y 122.541,Z 344.503,A -85,B 0,C 180,E1 -27152.343,E2 -27152.343} C_VEL
LIN {X 0,Y 119.503,Z 336.398,A -85,B 0,C 180,E1 -27155.691,E2 -27155.691} C_VEL
LIN {X 0,Y 117.083,Z 330.773,A -85,B 0,C 180,E1 -27158.66,E2 -27158.66} C_VEL
LIN {X 0,Y 114.901,Z 327.358,A -85,B 0,C 180,E1 -27161.501,E2 -27161.501} C_VEL
LIN {X 0,Y 112.167,Z 323.217,A -85,B 0,C 180,E1 -27165.776,E2 -27165.776} C_VEL
LIN {X 0,Y 109.886,Z 320.134,A -85,B 0,C 180,E1 -27170.365,E2 -27170.365} C_VEL
LIN {X 0,Y 109.261,Z 318.58,A -85,B 0,C 180,E1 -27172.145,E2 -27172.145} C_VEL
LIN {X 0,Y 107.127,Z 316.199,A -85,B 0,C 180,E1 -27180.941,E2 -27180.941} C_VEL
LIN {X 0,Y 106.957,Z 316.451,A -85,B 0,C 180,E1 -27187.552,E2 -27187.552} C_VEL
LIN {X 0,Y 109.276,Z 318.936,A -85,B 0,C 180,E1 -27197.793,E2 -27197.793} C_VEL
LIN {X 0,Y 110.933,Z 322.162,A -85,B 0,C 180,E1 -27201.852,E2 -27201.852} C_VEL
LIN {X 0,Y 112.598,Z 324.003,A -85,B 0,C 180,E1 -27204.795,E2 -27204.795} C_VEL
LIN {X 0,Y 115.6,Z 328.493,A -85,B 0,C 180,E1 -27209.259,E2 -27209.259} C_VEL
LIN {X 0,Y 118.582,Z 333.274,A -85,B 0,C 180,E1 -27212.898,E2 -27212.898} C_VEL
LIN {X 0,Y 121.987,Z 339.179,A -85,B 0,C 180,E1 -27216.453,E2 -27216.453} C_VEL
LIN {X 0,Y 125.527,Z 345.945,A -85,B 0,C 180,E1 -27219.69,E2 -27219.69} C_VEL
LIN {X 0,Y 128.577,Z 352.7,A -85,B 0,C 180,E1 -27222.234,E2 -27222.234} C_VEL
LIN {X 0,Y 126.443,Z 381.431,A -85,B 0,C 180,E1 -27223.736,E2 -27223.736} C_VEL
LIN {X 0,Y 124.699,Z 394.215,A -85,B 0,C 180,E1 -27224.927,E2 -27224.927} C_VEL
LIN {X 0,Y 121.992,Z 406.696,A -85,B 0,C 180,E1 -27226.553,E2 -27226.553} C_VEL
LIN {X 0,Y 118.409,Z 418.649,A -85,B 0,C 180,E1 -27228.68,E2 -27228.68} C_VEL
LIN {X 0,Y 114.152,Z 430.013,A -85,B 0,C 180,E1 -27231.441,E2 -27231.441} C_VEL
LIN {X 0,Y 109.583,Z 440.263,A -85,B 0,C 180,E1 -27234.748,E2 -27234.748} C_VEL
LIN {X 0,Y 104.784,Z 449.517,A -85,B 0,C 180,E1 -27238.684,E2 -27238.684} C_VEL
LIN {X 0,Y 99.617,Z 458.458,A -85,B 0,C 180,E1 -27243.839,E2 -27243.839} C_VEL
LIN {X 0,Y 95.203,Z 465.675,A -85,B 0,C 180,E1 -27249.475,E2 -27249.475} C_VEL
LIN {X 0,Y 91.212,Z 472.278,A -85,B 0,C 180,E1 -27256.637,E2 -27256.637} C_VEL
LIN {X 0,Y 88.683,Z 476.675,A -85,B 0,C 180,E1 -27263.175,E2 -27263.175} C_VEL
LIN {X 0,Y 87.076,Z 480.035,A -85,B 0,C 180,E1 -27270.002,E2 -27270.002} C_VEL
LIN {X 0,Y 86.767,Z 481.698,A -85,B 0,C 180,E1 -27274.648,E2 -27274.648} C_VEL
LIN {X 0,Y 86.88,Z 482.977,A -85,B 0,C 180,E1 -27279.312,E2 -27279.312} C_VEL
LIN {X 0,Y 87.837,Z 484.135,A -85,B 0,C 180,E1 -27286.225,E2 -27286.225} C_VEL
LIN {X 0,Y 89.842,Z 484.424,A -85,B 0,C 180,E1 -27293.026,E2 -27293.026} C_VEL
LIN {X 0,Y 91.757,Z 484.133,A -85,B 0,C 180,E1 -27297.36,E2 -27297.36} C_VEL
LIN {X 0,Y 94.127,Z 483.441,A -85,B 0,C 180,E1 -27301.512,E2 -27301.512} C_VEL
LIN {X 0,Y 100.126,Z 480.769,A -85,B 0,C 180,E1 -27309.179,E2 -27309.179} C_VEL
LIN {X 0,Y 105.543,Z 477.635,A -85,B 0,C 180,E1 -27314.363,E2 -27314.363} C_VEL
LIN {X 0,Y 111.66,Z 473.415,A -85,B 0,C 180,E1 -27319.052,E2 -27319.052} C_VEL
LIN {X 0,Y 118.795,Z 467.631,A -85,B 0,C 180,E1 -27323.498,E2 -27323.498} C_VEL
LIN {X 0,Y 125.615,Z 461.126,A -85,B 0,C 180,E1 -27327.06,E2 -27327.06} C_VEL
LIN {X 0,Y 133.281,Z 452.454,A -85,B 0,C 180,E1 -27330.465,E2 -27330.465} C_VEL
LIN {X 0,Y 139.919,Z 443.453,A -85,B 0,C 180,E1 -27333.123,E2 -27333.123} C_VEL
LIN {X 0,Y 146.006,Z 433.6,A -85,B 0,C 180,E1 -27335.305,E2 -27335.305} C_VEL
LIN {X 0,Y 151.557,Z 422.474,A -85,B 0,C 180,E1 -27337.167,E2 -27337.167} C_VEL
LIN {X 0,Y 156.336,Z 410.422,A -85,B 0,C 180,E1 -27338.646,E2 -27338.646} C_VEL
LIN {X 0,Y 159.968,Z 397.98,A -85,B 0,C 180,E1 -27339.789,E2 -27339.789} C_VEL
LIN {X 0,Y 162.326,Z 385.289,A -85,B 0,C 180,E1 -27340.704,E2 -27340.704} C_VEL
LIN {X 0,Y 162.704,Z 382.487,A -85,B 0,C 180,E1 -27340.88,E2 -27340.88} C_VEL
LIN {X 0,Y 160.047,Z 376.239,A -85,B 0,C 180,E1 -27344.273,E2 -27344.273} C_VEL
LIN {X 0,Y 157.581,Z 371.043,A -85,B 0,C 180,E1 -27347.932,E2 -27347.932} C_VEL
LIN {X 0,Y 156.391,Z 368.662,A -85,B 0,C 180,E1 -27350.073,E2 -27350.073} C_VEL
LIN {X 0,Y 154.928,Z 365.596,A -85,B 0,C 180,E1 -27353.406,E2 -27353.406} C_VEL
LIN {X 0,Y 153.46,Z 361.829,A -85,B 0,C 180,E1 -27359.343,E2 -27359.343} C_VEL
LIN {X 0,Y 153.364,Z 361.969,A -85,B 0,C 180,E1 -27366.578,E2 -27366.578} C_VEL
LIN {X 0,Y 153.571,Z 362.952,A -85,B 0,C 180,E1 -27368.222,E2 -27368.222} C_VEL
LIN {X 0,Y 154.704,Z 365.858,A -85,B 0,C 180,E1 -27372.578,E2 -27372.578} C_VEL
LIN {X 0,Y 156.526,Z 372.135,A -85,B 0,C 180,E1 -27377.199,E2 -27377.199} C_VEL
LIN {X 0,Y 158.081,Z 377.489,A -85,B 0,C 180,E1 -27380.134,E2 -27380.134} C_VEL
LIN {X 0,Y 160.124,Z 384.994,A -85,B 0,C 180,E1 -27383.341,E2 -27383.341} C_VEL
LIN {X 0,Y 161.191,Z 389.384,A -85,B 0,C 180,E1 -27384.864,E2 -27384.864} C_VEL
LIN {X 0,Y 160.602,Z 399.779,A -85,B 0,C 180,E1 -27385.828,E2 -27385.828} C_VEL
LIN {X 0,Y 157.908,Z 412.651,A -85,B 0,C 180,E1 -27386.427,E2 -27386.427} C_VEL
LIN {X 0,Y 154.223,Z 424.548,A -85,B 0,C 180,E1 -27387.183,E2 -27387.183} C_VEL
LIN {X 0,Y 149.576,Z 435.979,A -85,B 0,C 180,E1 -27388.238,E2 -27388.238} C_VEL
LIN {X 0,Y 143.656,Z 447.574,A -85,B 0,C 180,E1 -27389.73,E2 -27389.73} C_VEL
LIN {X 0,Y 136.984,Z 458.038,A -85,B 0,C 180,E1 -27391.466,E2 -27391.466} C_VEL
LIN {X 0,Y 130.531,Z 466.622,A -85,B 0,C 180,E1 -27393.431,E2 -27393.431} C_VEL
LIN {X 0,Y 123.646,Z 474.577,A -85,B 0,C 180,E1 -27395.907,E2 -27395.907} C_VEL
LIN {X 0,Y 115.828,Z 482.4,A -85,B 0,C 180,E1 -27399.319,E2 -27399.319} C_VEL
LIN {X 0,Y 107.469,Z 489.674,A -85,B 0,C 180,E1 -27403.998,E2 -27403.998} C_VEL
LIN {X 0,Y 101.097,Z 494.591,A -85,B 0,C 180,E1 -27408.668,E2 -27408.668} C_VEL
LIN {X 0,Y 94.733,Z 499.009,A -85,B 0,C 180,E1 -27414.941,E2 -27414.941} C_VEL
LIN {X 0,Y 89.879,Z 502.057,A -85,B 0,C 180,E1 -27422.018,E2 -27422.018} C_VEL
LIN {X 0,Y 86.353,Z 504.07,A -85,B 0,C 180,E1 -27431,E2 -27431} C_VEL
LIN {X 0,Y 85.273,Z 504.583,A -85,B 0,C 180,E1 -27440.511,E2 -27440.511} C_VEL
LIN {X 0,Y 85.584,Z 504.225,A -85,B 0,C 180,E1 -27445.288,E2 -27445.288} C_VEL
LIN {X 0,Y 86.004,Z 503.427,A -85,B 0,C 180,E1 -27449.998,E2 -27449.998} C_VEL
LIN {X 0,Y 85.177,Z 500.754,A -85,B 0,C 180,E1 -27458.064,E2 -27458.064} C_VEL
LIN {X 0,Y 85.77,Z 496.472,A -85,B 0,C 180,E1 -27466.663,E2 -27466.663} C_VEL
LIN {X 0,Y 87.634,Z 491.65,A -85,B 0,C 180,E1 -27473.637,E2 -27473.637} C_VEL
LIN {X 0,Y 91.568,Z 484.444,A -85,B 0,C 180,E1 -27481.2,E2 -27481.2} C_VEL
LIN {X 0,Y 96.197,Z 476.683,A -85,B 0,C 180,E1 -27487.063,E2 -27487.063} C_VEL
LIN {X 0,Y 100.697,Z 468.73,A -85,B 0,C 180,E1 -27491.529,E2 -27491.529} C_VEL
LIN {X 0,Y 105.95,Z 459.073,A -85,B 0,C 180,E1 -27495.483,E2 -27495.483} C_VEL
LIN {X 0,Y 111.079,Z 448.367,A -85,B 0,C 180,E1 -27498.702,E2 -27498.702} C_VEL
LIN {X 0,Y 115.325,Z 438.051,A -85,B 0,C 180,E1 -27500.983,E2 -27500.983} C_VEL
LIN {X 0,Y 119.454,Z 425.83,A -85,B 0,C 180,E1 -27502.93,E2 -27502.93} C_VEL
LIN {X 0,Y 122.665,Z 412.155,A -85,B 0,C 180,E1 -27504.532,E2 -27504.532} C_VEL
LIN {X 0,Y 124.757,Z 399.253,A -85,B 0,C 180,E1 -27505.47,E2 -27505.47} C_VEL
LIN {X 0,Y 125.541,Z 389.246,A -85,B 0,C 180,E1 -27506.018,E2 -27506.018} C_VEL
LIN {X 0,Y 125.717,Z 359.454,A -85,B 0,C 180,E1 -27508.672,E2 -27508.672} C_VEL
LIN {X 0,Y 125.645,Z 354.286,A -85,B 0,C 180,E1 -27509.215,E2 -27509.215} C_VEL
LIN {X 0,Y 125.533,Z 353.946,A -85,B 0,C 180,E1 -27509.32,E2 -27509.32} C_VEL
LIN {X 0,Y 124.334,Z 351.048,A -85,B 0,C 180,E1 -27510.396,E2 -27510.396} C_VEL
LIN {X 0,Y 122.727,Z 348.863,A -85,B 0,C 180,E1 -27511.742,E2 -27511.742} C_VEL
LIN {X 0,Y 117.635,Z 343.616,A -85,B 0,C 180,E1 -27516.446,E2 -27516.446} C_VEL
LIN {X 0,Y 117.177,Z 342.87,A -85,B 0,C 180,E1 -27516.961,E2 -27516.961} C_VEL
LIN {X 0,Y 115.032,Z 337.359,A -85,B 0,C 180,E1 -27519.852,E2 -27519.852} C_VEL
LIN {X 0,Y 112.881,Z 333.57,A -85,B 0,C 180,E1 -27522.945,E2 -27522.945} C_VEL
LIN {X 0,Y 110.591,Z 329.838,A -85,B 0,C 180,E1 -27526.877,E2 -27526.877} C_VEL
LIN {X 0,Y 108.467,Z 326.673,A -85,B 0,C 180,E1 -27531.618,E2 -27531.618} C_VEL
LIN {X 0,Y 108.042,Z 325.453,A -85,B 0,C 180,E1 -27532.995,E2 -27532.995} C_VEL
LIN {X 0,Y 106.252,Z 323.273,A -85,B 0,C 180,E1 -27540.948,E2 -27540.948} C_VEL
LIN {X 0,Y 106.06,Z 323.465,A -85,B 0,C 180,E1 -27547.149,E2 -27547.149} C_VEL
LIN {X 0,Y 108.027,Z 325.842,A -85,B 0,C 180,E1 -27556.885,E2 -27556.885} C_VEL
LIN {X 0,Y 109.752,Z 329.139,A -85,B 0,C 180,E1 -27561.359,E2 -27561.359} C_VEL
LIN {X 0,Y 110.981,Z 330.652,A -85,B 0,C 180,E1 -27563.698,E2 -27563.698} C_VEL
LIN {X 0,Y 113.716,Z 335.047,A -85,B 0,C 180,E1 -27568.117,E2 -27568.117} C_VEL
LIN {X 0,Y 116.216,Z 339.302,A -85,B 0,C 180,E1 -27571.44,E2 -27571.44} C_VEL
LIN {X 0,Y 118.714,Z 343.789,A -85,B 0,C 180,E1 -27574.323,E2 -27574.323} C_VEL
LIN {X 0,Y 122.134,Z 350.711,A -85,B 0,C 180,E1 -27577.822,E2 -27577.822} C_VEL
LIN {X 0,Y 124.223,Z 355.635,A -85,B 0,C 180,E1 -27579.788,E2 -27579.788} C_VEL
LIN {X 0,Y 121.93,Z 383.308,A -85,B 0,C 180,E1 -27581.242,E2 -27581.242} C_VEL
LIN {X 0,Y 119.94,Z 396.667,A -85,B 0,C 180,E1 -27582.567,E2 -27582.567} C_VEL
LIN {X 0,Y 117.015,Z 408.801,A -85,B 0,C 180,E1 -27584.198,E2 -27584.198} C_VEL
LIN {X 0,Y 113.251,Z 420.419,A -85,B 0,C 180,E1 -27586.343,E2 -27586.343} C_VEL
LIN {X 0,Y 108.768,Z 431.612,A -85,B 0,C 180,E1 -27589.143,E2 -27589.143} C_VEL
LIN {X 0,Y 103.924,Z 441.731,A -85,B 0,C 180,E1 -27592.512,E2 -27592.512} C_VEL
LIN {X 0,Y 98.848,Z 450.84,A -85,B 0,C 180,E1 -27596.566,E2 -27596.566} C_VEL
LIN {X 0,Y 93.344,Z 459.705,A -85,B 0,C 180,E1 -27601.931,E2 -27601.931} C_VEL
LIN {X 0,Y 88.649,Z 466.849,A -85,B 0,C 180,E1 -27607.881,E2 -27607.881} C_VEL
LIN {X 0,Y 85.534,Z 471.658,A -85,B 0,C 180,E1 -27613.289,E2 -27613.289} C_VEL
LIN {X 0,Y 82.453,Z 476.385,A -85,B 0,C 180,E1 -27620.187,E2 -27620.187} C_VEL
LIN {X 0,Y 80.436,Z 480.026,A -85,B 0,C 180,E1 -27627.498,E2 -27627.498} C_VEL
LIN {X 0,Y 79.719,Z 482.656,A -85,B 0,C 180,E1 -27635.06,E2 -27635.06} C_VEL
LIN {X 0,Y 79.89,Z 483.913,A -85,B 0,C 180,E1 -27640.135,E2 -27640.135} C_VEL
LIN {X 0,Y 80.909,Z 484.975,A -85,B 0,C 180,E1 -27647.154,E2 -27647.154} C_VEL
LIN {X 0,Y 83.34,Z 485.268,A -85,B 0,C 180,E1 -27654.94,E2 -27654.94} C_VEL
LIN {X 0,Y 85.492,Z 484.955,A -85,B 0,C 180,E1 -27659.555,E2 -27659.555} C_VEL
LIN {X 0,Y 88.11,Z 484.218,A -85,B 0,C 180,E1 -27663.943,E2 -27663.943} C_VEL
LIN {X 0,Y 94.687,Z 481.497,A -85,B 0,C 180,E1 -27671.915,E2 -27671.915} C_VEL
LIN {X 0,Y 100.557,Z 478.31,A -85,B 0,C 180,E1 -27677.212,E2 -27677.212} C_VEL
LIN {X 0,Y 107.099,Z 474.036,A -85,B 0,C 180,E1 -27681.949,E2 -27681.949} C_VEL
LIN {X 0,Y 114.333,Z 468.476,A -85,B 0,C 180,E1 -27686.179,E2 -27686.179} C_VEL
LIN {X 0,Y 121.869,Z 461.587,A -85,B 0,C 180,E1 -27689.886,E2 -27689.886} C_VEL
LIN {X 0,Y 129.902,Z 452.828,A -85,B 0,C 180,E1 -27693.213,E2 -27693.213} C_VEL
LIN {X 0,Y 136.452,Z 444.256,A -85,B 0,C 180,E1 -27695.666,E2 -27695.666} C_VEL
LIN {X 0,Y 143.154,Z 433.697,A -85,B 0,C 180,E1 -27697.918,E2 -27697.918} C_VEL
LIN {X 0,Y 148.92,Z 422.384,A -85,B 0,C 180,E1 -27699.712,E2 -27699.712} C_VEL
LIN {X 0,Y 153.524,Z 411.003,A -85,B 0,C 180,E1 -27701.047,E2 -27701.047} C_VEL
LIN {X 0,Y 157.208,Z 398.688,A -85,B 0,C 180,E1 -27702.145,E2 -27702.145} C_VEL
LIN {X 0,Y 159.582,Z 386.37,A -85,B 0,C 180,E1 -27703.035,E2 -27703.035} C_VEL
LIN {X 0,Y 157.714,Z 381.278,A -85,B 0,C 180,E1 -27706.059,E2 -27706.059} C_VEL
LIN {X 0,Y 155.541,Z 376.192,A -85,B 0,C 180,E1 -27709.916,E2 -27709.916} C_VEL
LIN {X 0,Y 153.77,Z 372.377,A -85,B 0,C 180,E1 -27714.097,E2 -27714.097} C_VEL
LIN {X 0,Y 152.494,Z 368.775,A -85,B 0,C 180,E1 -27719.999,E2 -27719.999} C_VEL
LIN {X 0,Y 152.514,Z 369.181,A -85,B 0,C 180,E1 -27726.808,E2 -27726.808} C_VEL
LIN {X 0,Y 153.596,Z 372.741,A -85,B 0,C 180,E1 -27732,E2 -27732} C_VEL
LIN {X 0,Y 155.021,Z 378.437,A -85,B 0,C 180,E1 -27736.116,E2 -27736.116} C_VEL
LIN {X 0,Y 156.492,Z 384.16,A -85,B 0,C 180,E1 -27739.235,E2 -27739.235} C_VEL
LIN {X 0,Y 158.12,Z 391.213,A -85,B 0,C 180,E1 -27742.16,E2 -27742.16} C_VEL
LIN {X 0,Y 158.433,Z 393.275,A -85,B 0,C 180,E1 -27742.802,E2 -27742.802} C_VEL
LIN {X 0,Y 157.769,Z 400.704,A -85,B 0,C 180,E1 -27743.492,E2 -27743.492} C_VEL
LIN {X 0,Y 154.919,Z 413.295,A -85,B 0,C 180,E1 -27744.078,E2 -27744.078} C_VEL
LIN {X 0,Y 150.757,Z 425.722,A -85,B 0,C 180,E1 -27744.866,E2 -27744.866} C_VEL
LIN {X 0,Y 145.604,Z 437.563,A -85,B 0,C 180,E1 -27745.975,E2 -27745.975} C_VEL
LIN {X 0,Y 139.52,Z 448.71,A -85,B 0,C 180,E1 -27747.4,E2 -27747.4} C_VEL
LIN {X 0,Y 132.671,Z 458.759,A -85,B 0,C 180,E1 -27749.067,E2 -27749.067} C_VEL
LIN {X 0,Y 125.314,Z 467.899,A -85,B 0,C 180,E1 -27751.21,E2 -27751.21} C_VEL
LIN {X 0,Y 116.839,Z 476.86,A -85,B 0,C 180,E1 -27754.199,E2 -27754.199} C_VEL
LIN {X 0,Y 108.864,Z 484.114,A -85,B 0,C 180,E1 -27757.736,E2 -27757.736} C_VEL
LIN {X 0,Y 100.282,Z 490.794,A -85,B 0,C 180,E1 -27762.619,E2 -27762.619} C_VEL
LIN {X 0,Y 93.763,Z 495.288,A -85,B 0,C 180,E1 -27767.576,E2 -27767.576} C_VEL
LIN {X 0,Y 89.428,Z 498.01,A -85,B 0,C 180,E1 -27771.801,E2 -27771.801} C_VEL
LIN {X 0,Y 83.639,Z 501.272,A -85,B 0,C 180,E1 -27779.723,E2 -27779.723} C_VEL
LIN {X 0,Y 79.626,Z 503.241,A -85,B 0,C 180,E1 -27789.324,E2 -27789.324} C_VEL
LIN {X 0,Y 78.598,Z 503.671,A -85,B 0,C 180,E1 -27794.438,E2 -27794.438} C_VEL
LIN {X 0,Y 78.508,Z 503.316,A -85,B 0,C 180,E1 -27804.862,E2 -27804.862} C_VEL
LIN {X 0,Y 78.899,Z 502.496,A -85,B 0,C 180,E1 -27809.998,E2 -27809.998} C_VEL
LIN {X 0,Y 78.124,Z 499.957,A -85,B 0,C 180,E1 -27818.293,E2 -27818.293} C_VEL
LIN {X 0,Y 78.484,Z 496.765,A -85,B 0,C 180,E1 -27825.581,E2 -27825.581} C_VEL
LIN {X 0,Y 80.231,Z 492.285,A -85,B 0,C 180,E1 -27833.213,E2 -27833.213} C_VEL
LIN {X 0,Y 83.362,Z 486.603,A -85,B 0,C 180,E1 -27840.384,E2 -27840.384} C_VEL
LIN {X 0,Y 88.187,Z 479.156,A -85,B 0,C 180,E1 -27847.162,E2 -27847.162} C_VEL
LIN {X 0,Y 93.422,Z 470.768,A -85,B 0,C 180,E1 -27852.61,E2 -27852.61} C_VEL
LIN {X 0,Y 98.709,Z 461.756,A -85,B 0,C 180,E1 -27856.865,E2 -27856.865} C_VEL
LIN {X 0,Y 103.417,Z 453.096,A -85,B 0,C 180,E1 -27859.861,E2 -27859.861} C_VEL
LIN {X 0,Y 108.442,Z 442.586,A -85,B 0,C 180,E1 -27862.548,E2 -27862.548} C_VEL
LIN {X 0,Y 112.997,Z 431.013,A -85,B 0,C 180,E1 -27864.714,E2 -27864.714} C_VEL
LIN {X 0,Y 116.556,Z 418.937,A -85,B 0,C 180,E1 -27866.389,E2 -27866.389} C_VEL
LIN {X 0,Y 119.424,Z 405.338,A -85,B 0,C 180,E1 -27867.681,E2 -27867.681} C_VEL
LIN {X 0,Y 121.134,Z 391.834,A -85,B 0,C 180,E1 -27868.444,E2 -27868.444} C_VEL
LIN {X 0,Y 121.614,Z 361.069,A -85,B 0,C 180,E1 -27871.251,E2 -27871.251} C_VEL
LIN {X 0,Y 121.494,Z 356.65,A -85,B 0,C 180,E1 -27871.806,E2 -27871.806} C_VEL
LIN {X 0,Y 118.7,Z 347.39,A -85,B 0,C 180,E1 -27875.049,E2 -27875.049} C_VEL
LIN {X 0,Y 117.177,Z 342.87,A -85,B 0,C 180,E1 -27876.961,E2 -27876.961} C_VEL
LIN {X 0,Y 115.129,Z 340.152,A -85,B 0,C 180,E1 -27879.348,E2 -27879.348} C_VEL
LIN {X 0,Y 112.98,Z 338.476,A -85,B 0,C 180,E1 -27882.014,E2 -27882.014} C_VEL
LIN {X 0,Y 108.21,Z 335.339,A -85,B 0,C 180,E1 -27889.841,E2 -27889.841} C_VEL
LIN {X 0,Y 107.446,Z 334.019,A -85,B 0,C 180,E1 -27891.824,E2 -27891.824} C_VEL
LIN {X 0,Y 106.775,Z 332.245,A -85,B 0,C 180,E1 -27894.098,E2 -27894.098} C_VEL
LIN {X 0,Y 105.259,Z 330.277,A -85,B 0,C 180,E1 -27902.152,E2 -27902.152} C_VEL
LIN {X 0,Y 105.29,Z 330.719,A -85,B 0,C 180,E1 -27908.476,E2 -27908.476} C_VEL
LIN {X 0,Y 106.794,Z 332.664,A -85,B 0,C 180,E1 -27915.894,E2 -27915.894} C_VEL
LIN {X 0,Y 108.576,Z 336.137,A -85,B 0,C 180,E1 -27920.856,E2 -27920.856} C_VEL
LIN {X 0,Y 109.454,Z 337.358,A -85,B 0,C 180,E1 -27922.661,E2 -27922.661} C_VEL
LIN {X 0,Y 111.65,Z 341.129,A -85,B 0,C 180,E1 -27926.566,E2 -27926.566} C_VEL
LIN {X 0,Y 114.641,Z 346.505,A -85,B 0,C 180,E1 -27930.846,E2 -27930.846} C_VEL
LIN {X 0,Y 118.546,Z 354.655,A -85,B 0,C 180,E1 -27935.482,E2 -27935.482} C_VEL
LIN {X 0,Y 120.038,Z 358.236,A -85,B 0,C 180,E1 -27937.076,E2 -27937.076} C_VEL
LIN {X 0,Y 117.931,Z 383.325,A -85,B 0,C 180,E1 -27938.441,E2 -27938.441} C_VEL
LIN {X 0,Y 115.818,Z 396.897,A -85,B 0,C 180,E1 -27939.755,E2 -27939.755} C_VEL
LIN {X 0,Y 112.559,Z 409.833,A -85,B 0,C 180,E1 -27941.478,E2 -27941.478} C_VEL
LIN {X 0,Y 108.295,Z 422.19,A -85,B 0,C 180,E1 -27943.786,E2 -27943.786} C_VEL
LIN {X 0,Y 103.574,Z 433.212,A -85,B 0,C 180,E1 -27946.608,E2 -27946.608} C_VEL
LIN {X 0,Y 98.442,Z 443.162,A -85,B 0,C 180,E1 -27950.023,E2 -27950.023} C_VEL
LIN {X 0,Y 93.064,Z 452.163,A -85,B 0,C 180,E1 -27954.182,E2 -27954.182} C_VEL
LIN {X 0,Y 87.192,Z 460.951,A -85,B 0,C 180,E1 -27959.753,E2 -27959.753} C_VEL
LIN {X 0,Y 82.174,Z 468.014,A -85,B 0,C 180,E1 -27966.033,E2 -27966.033} C_VEL
LIN {X 0,Y 77.557,Z 474.449,A -85,B 0,C 180,E1 -27974.228,E2 -27974.228} C_VEL
LIN {X 0,Y 74.659,Z 478.742,A -85,B 0,C 180,E1 -27981.885,E2 -27981.885} C_VEL
LIN {X 0,Y 72.923,Z 482,A -85,B 0,C 180,E1 -27990.002,E2 -27990.002} C_VEL
LIN {X 0,Y 72.676,Z 483.614,A -85,B 0,C 180,E1 -27995.552,E2 -27995.552} C_VEL
LIN {X 0,Y 72.92,Z 484.846,A -85,B 0,C 180,E1 -28001.116,E2 -28001.116} C_VEL
LIN {X 0,Y 75.006,Z 486.075,A -85,B 0,C 180,E1 -28012.014,E2 -28012.014} C_VEL
LIN {X 0,Y 79.358,Z 485.773,A -85,B 0,C 180,E1 -28022.099,E2 -28022.099} C_VEL
LIN {X 0,Y 82.278,Z 484.994,A -85,B 0,C 180,E1 -28026.723,E2 -28026.723} C_VEL
LIN {X 0,Y 85.711,Z 483.806,A -85,B 0,C 180,E1 -28030.995,E2 -28030.995} C_VEL
LIN {X 0,Y 89.706,Z 482.136,A -85,B 0,C 180,E1 -28035.16,E2 -28035.16} C_VEL
LIN {X 0,Y 95.84,Z 478.986,A -85,B 0,C 180,E1 -28040.352,E2 -28040.352} C_VEL
LIN {X 0,Y 102.848,Z 474.655,A -85,B 0,C 180,E1 -28045.087,E2 -28045.087} C_VEL
LIN {X 0,Y 111.264,Z 468.394,A -85,B 0,C 180,E1 -28049.646,E2 -28049.646} C_VEL
LIN {X 0,Y 119.816,Z 460.702,A -85,B 0,C 180,E1 -28053.447,E2 -28053.447} C_VEL
LIN {X 0,Y 126.831,Z 453.203,A -85,B 0,C 180,E1 -28056.108,E2 -28056.108} C_VEL
LIN {X 0,Y 133.313,Z 445.004,A -85,B 0,C 180,E1 -28058.344,E2 -28058.344} C_VEL
LIN {X 0,Y 139.87,Z 435.078,A -85,B 0,C 180,E1 -28060.411,E2 -28060.411} C_VEL
LIN {X 0,Y 145.831,Z 423.893,A -85,B 0,C 180,E1 -28062.139,E2 -28062.139} C_VEL
LIN {X 0,Y 150.643,Z 412.539,A -85,B 0,C 180,E1 -28063.43,E2 -28063.43} C_VEL
LIN {X 0,Y 154.364,Z 400.933,A -85,B 0,C 180,E1 -28064.433,E2 -28064.433} C_VEL
LIN {X 0,Y 156.651,Z 390.288,A -85,B 0,C 180,E1 -28065.282,E2 -28065.282} C_VEL
LIN {X 0,Y 154.747,Z 384.448,A -85,B 0,C 180,E1 -28069.367,E2 -28069.367} C_VEL
LIN {X 0,Y 153.628,Z 381.688,A -85,B 0,C 180,E1 -28071.946,E2 -28071.946} C_VEL
LIN {X 0,Y 152.663,Z 379.188,A -85,B 0,C 180,E1 -28074.717,E2 -28074.717} C_VEL
LIN {X 0,Y 151.624,Z 375.832,A -85,B 0,C 180,E1 -28079.999,E2 -28079.999} C_VEL
LIN {X 0,Y 151.579,Z 376.14,A -85,B 0,C 180,E1 -28086.322,E2 -28086.322} C_VEL
LIN {X 0,Y 152.43,Z 379.354,A -85,B 0,C 180,E1 -28091.132,E2 -28091.132} C_VEL
LIN {X 0,Y 153.551,Z 384.693,A -85,B 0,C 180,E1 -28094.965,E2 -28094.965} C_VEL
LIN {X 0,Y 154.673,Z 389.766,A -85,B 0,C 180,E1 -28097.775,E2 -28097.775} C_VEL
LIN {X 0,Y 155.793,Z 395.995,A -85,B 0,C 180,E1 -28100.448,E2 -28100.448} C_VEL
LIN {X 0,Y 155.771,Z 397.266,A -85,B 0,C 180,E1 -28100.716,E2 -28100.716} C_VEL
LIN {X 0,Y 154.997,Z 402.593,A -85,B 0,C 180,E1 -28101.135,E2 -28101.135} C_VEL
LIN {X 0,Y 151.365,Z 416.458,A -85,B 0,C 180,E1 -28101.78,E2 -28101.78} C_VEL
LIN {X 0,Y 146.802,Z 428.732,A -85,B 0,C 180,E1 -28102.608,E2 -28102.608} C_VEL
LIN {X 0,Y 141.089,Z 440.508,A -85,B 0,C 180,E1 -28103.751,E2 -28103.751} C_VEL
LIN {X 0,Y 134.065,Z 452.051,A -85,B 0,C 180,E1 -28105.273,E2 -28105.273} C_VEL
LIN {X 0,Y 126.305,Z 462.274,A -85,B 0,C 180,E1 -28107.09,E2 -28107.09} C_VEL
LIN {X 0,Y 118.82,Z 470.655,A -85,B 0,C 180,E1 -28109.257,E2 -28109.257} C_VEL
LIN {X 0,Y 110.183,Z 478.906,A -85,B 0,C 180,E1 -28112.312,E2 -28112.312} C_VEL
LIN {X 0,Y 101.979,Z 485.598,A -85,B 0,C 180,E1 -28115.926,E2 -28115.926} C_VEL
LIN {X 0,Y 93.198,Z 491.766,A -85,B 0,C 180,E1 -28121.052,E2 -28121.052} C_VEL
LIN {X 0,Y 86.489,Z 495.858,A -85,B 0,C 180,E1 -28126.313,E2 -28126.313} C_VEL
LIN {X 0,Y 80.75,Z 498.96,A -85,B 0,C 180,E1 -28132.464,E2 -28132.464} C_VEL
LIN {X 0,Y 74.904,Z 501.631,A -85,B 0,C 180,E1 -28142.02,E2 -28142.02} C_VEL
LIN {X 0,Y 71.726,Z 502.811,A -85,B 0,C 180,E1 -28152.903,E2 -28152.903} C_VEL
LIN {X 0,Y 71.432,Z 502.406,A -85,B 0,C 180,E1 -28164.351,E2 -28164.351} C_VEL
LIN {X 0,Y 71.794,Z 501.565,A -85,B 0,C 180,E1 -28169.998,E2 -28169.998} C_VEL
LIN {X 0,Y 71.053,Z 499.191,A -85,B 0,C 180,E1 -28178.467,E2 -28178.467} C_VEL
LIN {X 0,Y 71.597,Z 495.733,A -85,B 0,C 180,E1 -28187.124,E2 -28187.124} C_VEL
LIN {X 0,Y 73.675,Z 491.201,A -85,B 0,C 180,E1 -28195.418,E2 -28195.418} C_VEL
LIN {X 0,Y 77.269,Z 485.469,A -85,B 0,C 180,E1 -28203.071,E2 -28203.071} C_VEL
LIN {X 0,Y 82.635,Z 477.864,A -85,B 0,C 180,E1 -28210.218,E2 -28210.218} C_VEL
LIN {X 0,Y 88.28,Z 469.463,A -85,B 0,C 180,E1 -28215.762,E2 -28215.762} C_VEL
LIN {X 0,Y 94.602,Z 459.387,A -85,B 0,C 180,E1 -28220.418,E2 -28220.418} C_VEL
LIN {X 0,Y 100.301,Z 449.178,A -85,B 0,C 180,E1 -28223.683,E2 -28223.683} C_VEL
LIN {X 0,Y 105.562,Z 437.811,A -85,B 0,C 180,E1 -28226.322,E2 -28226.322} C_VEL
LIN {X 0,Y 110.05,Z 426.068,A -85,B 0,C 180,E1 -28228.224,E2 -28228.224} C_VEL
LIN {X 0,Y 113.578,Z 413.19,A -85,B 0,C 180,E1 -28229.805,E2 -28229.805} C_VEL
LIN {X 0,Y 116.21,Z 399.309,A -85,B 0,C 180,E1 -28230.853,E2 -28230.853} C_VEL
LIN {X 0,Y 117.101,Z 390.262,A -85,B 0,C 180,E1 -28231.398,E2 -28231.398} C_VEL
LIN {X 0,Y 117.788,Z 361.424,A -85,B 0,C 180,E1 -28234.139,E2 -28234.139} C_VEL
LIN {X 0,Y 117.709,Z 359.422,A -85,B 0,C 180,E1 -28234.442,E2 -28234.442} C_VEL
LIN {X 0,Y 115.278,Z 350.802,A -85,B 0,C 180,E1 -28237.721,E2 -28237.721} C_VEL
LIN {X 0,Y 112.971,Z 343.849,A -85,B 0,C 180,E1 -28241.173,E2 -28241.173} C_VEL
LIN {X 0,Y 111.435,Z 340.482,A -85,B 0,C 180,E1 -28243.631,E2 -28243.631} C_VEL
LIN {X 0,Y 108.991,Z 336.389,A -85,B 0,C 180,E1 -28248.14,E2 -28248.14} C_VEL
LIN {X 0,Y 107.446,Z 334.019,A -85,B 0,C 180,E1 -28251.824,E2 -28251.824} C_VEL
LIN {X 0,Y 106.787,Z 332.982,A -85,B 0,C 180,E1 -28253.808,E2 -28253.808} C_VEL
LIN {X 0,Y 106.136,Z 332.741,A -85,B 0,C 180,E1 -28255.887,E2 -28255.887} C_VEL
LIN {X 0,Y 105.289,Z 333.446,A -85,B 0,C 180,E1 -28259.069,E2 -28259.069} C_VEL
LIN {X 0,Y 104.344,Z 337.16,A -85,B 0,C 180,E1 -28266.701,E2 -28266.701} C_VEL
LIN {X 0,Y 104.454,Z 337.941,A -85,B 0,C 180,E1 -28268.937,E2 -28268.937} C_VEL
LIN {X 0,Y 105.643,Z 339.634,A -85,B 0,C 180,E1 -28275.093,E2 -28275.093} C_VEL
LIN {X 0,Y 107.444,Z 343.153,A -85,B 0,C 180,E1 -28280.415,E2 -28280.415} C_VEL
LIN {X 0,Y 109.812,Z 347.49,A -85,B 0,C 180,E1 -28285.215,E2 -28285.215} C_VEL
LIN {X 0,Y 112.504,Z 352.798,A -85,B 0,C 180,E1 -28289.472,E2 -28289.472} C_VEL
LIN {X 0,Y 115.687,Z 360.022,A -85,B 0,C 180,E1 -28293.667,E2 -28293.667} C_VEL
LIN {X 0,Y 116.213,Z 361.413,A -85,B 0,C 180,E1 -28294.312,E2 -28294.312} C_VEL
LIN {X 0,Y 113.98,Z 385.223,A -85,B 0,C 180,E1 -28295.594,E2 -28295.594} C_VEL
LIN {X 0,Y 111.665,Z 398.809,A -85,B 0,C 180,E1 -28296.945,E2 -28296.945} C_VEL
LIN {X 0,Y 108.582,Z 410.27,A -85,B 0,C 180,E1 -28298.453,E2 -28298.453} C_VEL
LIN {X 0,Y 104.214,Z 422.401,A -85,B 0,C 180,E1 -28300.656,E2 -28300.656} C_VEL
LIN {X 0,Y 99.22,Z 433.538,A -85,B 0,C 180,E1 -28303.449,E2 -28303.449} C_VEL
LIN {X 0,Y 93.77,Z 443.609,A -85,B 0,C 180,E1 -28306.854,E2 -28306.854} C_VEL
LIN {X 0,Y 87.462,Z 453.487,A -85,B 0,C 180,E1 -28311.487,E2 -28311.487} C_VEL
LIN {X 0,Y 81.187,Z 462.196,A -85,B 0,C 180,E1 -28317.249,E2 -28317.249} C_VEL
LIN {X 0,Y 75.784,Z 469.164,A -85,B 0,C 180,E1 -28323.867,E2 -28323.867} C_VEL
LIN {X 0,Y 70.798,Z 475.534,A -85,B 0,C 180,E1 -28332.677,E2 -28332.677} C_VEL
LIN {X 0,Y 67.667,Z 479.776,A -85,B 0,C 180,E1 -28341.04,E2 -28341.04} C_VEL
LIN {X 0,Y 65.848,Z 482.983,A -85,B 0,C 180,E1 -28350.003,E2 -28350.003} C_VEL
LIN {X 0,Y 65.641,Z 484.571,A -85,B 0,C 180,E1 -28356.149,E2 -28356.149} C_VEL
LIN {X 0,Y 65.956,Z 485.77,A -85,B 0,C 180,E1 -28362.307,E2 -28362.307} C_VEL
LIN {X 0,Y 68.445,Z 486.945,A -85,B 0,C 180,E1 -28374.252,E2 -28374.252} C_VEL
LIN {X 0,Y 70.667,Z 486.96,A -85,B 0,C 180,E1 -28379.821,E2 -28379.821} C_VEL
LIN {X 0,Y 73.414,Z 486.579,A -85,B 0,C 180,E1 -28385.058,E2 -28385.058} C_VEL
LIN {X 0,Y 80.454,Z 484.558,A -85,B 0,C 180,E1 -28394.335,E2 -28394.335} C_VEL
LIN {X 0,Y 86.798,Z 481.948,A -85,B 0,C 180,E1 -28400.284,E2 -28400.284} C_VEL
LIN {X 0,Y 93.874,Z 478.306,A -85,B 0,C 180,E1 -28405.441,E2 -28405.441} C_VEL
LIN {X 0,Y 101.541,Z 473.52,A -85,B 0,C 180,E1 -28409.903,E2 -28409.903} C_VEL
LIN {X 0,Y 109.692,Z 467.436,A -85,B 0,C 180,E1 -28413.765,E2 -28413.765} C_VEL
LIN {X 0,Y 118.251,Z 459.766,A -85,B 0,C 180,E1 -28417.104,E2 -28417.104} C_VEL
LIN {X 0,Y 125.571,Z 451.871,A -85,B 0,C 180,E1 -28419.631,E2 -28419.631} C_VEL
LIN {X 0,Y 133.076,Z 442.171,A -85,B 0,C 180,E1 -28421.918,E2 -28421.918} C_VEL
LIN {X 0,Y 139.178,Z 432.602,A -85,B 0,C 180,E1 -28423.624,E2 -28423.624} C_VEL
LIN {X 0,Y 144.577,Z 422.243,A -85,B 0,C 180,E1 -28425.046,E2 -28425.046} C_VEL
LIN {X 0,Y 149.433,Z 410.3,A -85,B 0,C 180,E1 -28426.265,E2 -28426.265} C_VEL
LIN {X 0,Y 153.02,Z 398.221,A -85,B 0,C 180,E1 -28427.225,E2 -28427.225} C_VEL
LIN {X 0,Y 153.834,Z 394.496,A -85,B 0,C 180,E1 -28427.549,E2 -28427.549} C_VEL
LIN {X 0,Y 152.535,Z 389.359,A -85,B 0,C 180,E1 -28431.554,E2 -28431.554} C_VEL
LIN {X 0,Y 151.392,Z 385.804,A -85,B 0,C 180,E1 -28435.673,E2 -28435.673} C_VEL
LIN {X 0,Y 150.675,Z 382.87,A -85,B 0,C 180,E1 -28440.597,E2 -28440.597} C_VEL
LIN {X 0,Y 150.668,Z 383.194,A -85,B 0,C 180,E1 -28446.024,E2 -28446.024} C_VEL
LIN {X 0,Y 151.301,Z 386.049,A -85,B 0,C 180,E1 -28450.284,E2 -28450.284} C_VEL
LIN {X 0,Y 152.086,Z 390.902,A -85,B 0,C 180,E1 -28453.807,E2 -28453.807} C_VEL
LIN {X 0,Y 152.847,Z 396.018,A -85,B 0,C 180,E1 -28456.611,E2 -28456.611} C_VEL
LIN {X 0,Y 153.325,Z 399.946,A -85,B 0,C 180,E1 -28458.393,E2 -28458.393} C_VEL
LIN {X 0,Y 152.351,Z 404.921,A -85,B 0,C 180,E1 -28458.717,E2 -28458.717} C_VEL
LIN {X 0,Y 148.887,Z 417.011,A -85,B 0,C 180,E1 -28459.253,E2 -28459.253} C_VEL
LIN {X 0,Y 143.903,Z 429.545,A -85,B 0,C 180,E1 -28460.055,E2 -28460.055} C_VEL
LIN {X 0,Y 138.387,Z 440.437,A -85,B 0,C 180,E1 -28461.064,E2 -28461.064} C_VEL
LIN {X 0,Y 131.198,Z 451.824,A -85,B 0,C 180,E1 -28462.475,E2 -28462.475} C_VEL
LIN {X 0,Y 123.239,Z 461.902,A -85,B 0,C 180,E1 -28464.155,E2 -28464.155} C_VEL
LIN {X 0,Y 115.508,Z 470.198,A -85,B 0,C 180,E1 -28466.174,E2 -28466.174} C_VEL
LIN {X 0,Y 106.54,Z 478.38,A -85,B 0,C 180,E1 -28469.067,E2 -28469.067} C_VEL
LIN {X 0,Y 99.364,Z 483.977,A -85,B 0,C 180,E1 -28471.922,E2 -28471.922} C_VEL
LIN {X 0,Y 91.25,Z 489.514,A -85,B 0,C 180,E1 -28476.029,E2 -28476.029} C_VEL
LIN {X 0,Y 83.794,Z 493.906,A -85,B 0,C 180,E1 -28480.986,E2 -28480.986} C_VEL
LIN {X 0,Y 77.656,Z 497.032,A -85,B 0,C 180,E1 -28486.386,E2 -28486.386} C_VEL
LIN {X 0,Y 71.68,Z 499.705,A -85,B 0,C 180,E1 -28493.963,E2 -28493.963} C_VEL
LIN {X 0,Y 66.418,Z 501.583,A -85,B 0,C 180,E1 -28504.957,E2 -28504.957} C_VEL
LIN {X 0,Y 64.933,Z 501.944,A -85,B 0,C 180,E1 -28511.05,E2 -28511.05} C_VEL
LIN {X 0,Y 64.335,Z 501.493,A -85,B 0,C 180,E1 -28523.726,E2 -28523.726} C_VEL
LIN {X 0,Y 64.69,Z 500.635,A -85,B 0,C 180,E1 -28529.997,E2 -28529.997} C_VEL
LIN {X 0,Y 63.982,Z 498.428,A -85,B 0,C 180,E1 -28538.67,E2 -28538.67} C_VEL
LIN {X 0,Y 64.754,Z 494.698,A -85,B 0,C 180,E1 -28548.999,E2 -28548.999} C_VEL
LIN {X 0,Y 67.265,Z 490.119,A -85,B 0,C 180,E1 -28558.042,E2 -28558.042} C_VEL
LIN {X 0,Y 71.382,Z 484.336,A -85,B 0,C 180,E1 -28566.205,E2 -28566.205} C_VEL
LIN {X 0,Y 77.105,Z 476.938,A -85,B 0,C 180,E1 -28573.401,E2 -28573.401} C_VEL
LIN {X 0,Y 83.448,Z 468.161,A -85,B 0,C 180,E1 -28579.282,E2 -28579.282} C_VEL
LIN {X 0,Y 89.578,Z 458.989,A -85,B 0,C 180,E1 -28583.526,E2 -28583.526} C_VEL
LIN {X 0,Y 95.562,Z 448.917,A -85,B 0,C 180,E1 -28586.773,E2 -28586.773} C_VEL
LIN {X 0,Y 101.073,Z 437.691,A -85,B 0,C 180,E1 -28589.365,E2 -28589.365} C_VEL
LIN {X 0,Y 105.743,Z 426.134,A -85,B 0,C 180,E1 -28591.215,E2 -28591.215} C_VEL
LIN {X 0,Y 109.601,Z 412.965,A -85,B 0,C 180,E1 -28592.831,E2 -28592.831} C_VEL
LIN {X 0,Y 112.32,Z 399.659,A -85,B 0,C 180,E1 -28593.81,E2 -28593.81} C_VEL
LIN {X 0,Y 113.297,Z 391.017,A -85,B 0,C 180,E1 -28594.357,E2 -28594.357} C_VEL
LIN {X 0,Y 114.255,Z 362.874,A -85,B 0,C 180,E1 -28597.092,E2 -28597.092} C_VEL
LIN {X 0,Y 112.497,Z 355.686,A -85,B 0,C 180,E1 -28599.904,E2 -28599.904} C_VEL
LIN {X 0,Y 110.576,Z 349.176,A -85,B 0,C 180,E1 -28603.248,E2 -28603.248} C_VEL
LIN {X 0,Y 109.231,Z 346.219,A -85,B 0,C 180,E1 -28605.683,E2 -28605.683} C_VEL
LIN {X 0,Y 107.439,Z 342.9,A -85,B 0,C 180,E1 -28609.459,E2 -28609.459} C_VEL
LIN {X 0,Y 105.666,Z 339.31,A -85,B 0,C 180,E1 -28614.754,E2 -28614.754} C_VEL
LIN {X 0,Y 104.41,Z 337.327,A -85,B 0,C 180,E1 -28621.93,E2 -28621.93} C_VEL
LIN {X 0,Y 104.357,Z 337.67,A -85,B 0,C 180,E1 -28627.742,E2 -28627.742} C_VEL
LIN {X 0,Y 104.454,Z 337.941,A -85,B 0,C 180,E1 -28628.937,E2 -28628.937} C_VEL
LIN {X 0,Y 104.815,Z 339.502,A -85,B 0,C 180,E1 -28632.051,E2 -28632.051} C_VEL
LIN {X 0,Y 105.281,Z 342.155,A -85,B 0,C 180,E1 -28634.944,E2 -28634.944} C_VEL
LIN {X 0,Y 108.008,Z 353.756,A -85,B 0,C 180,E1 -28643.754,E2 -28643.754} C_VEL
LIN {X 0,Y 110.502,Z 359.238,A -85,B 0,C 180,E1 -28648.153,E2 -28648.153} C_VEL
LIN {X 0,Y 112.626,Z 364.488,A -85,B 0,C 180,E1 -28651.313,E2 -28651.313} C_VEL
LIN {X 0,Y 110.402,Z 386.513,A -85,B 0,C 180,E1 -28652.501,E2 -28652.501} C_VEL
LIN {X 0,Y 108.102,Z 399.241,A -85,B 0,C 180,E1 -28653.751,E2 -28653.751} C_VEL
LIN {X 0,Y 104.961,Z 410.551,A -85,B 0,C 180,E1 -28655.184,E2 -28655.184} C_VEL
LIN {X 0,Y 100.469,Z 422.601,A -85,B 0,C 180,E1 -28657.283,E2 -28657.283} C_VEL
LIN {X 0,Y 95.194,Z 433.858,A -85,B 0,C 180,E1 -28660.011,E2 -28660.011} C_VEL
LIN {X 0,Y 89.409,Z 444.037,A -85,B 0,C 180,E1 -28663.361,E2 -28663.361} C_VEL
LIN {X 0,Y 83.249,Z 453.202,A -85,B 0,C 180,E1 -28667.521,E2 -28667.521} C_VEL
LIN {X 0,Y 76.431,Z 462.098,A -85,B 0,C 180,E1 -28673.299,E2 -28673.299} C_VEL
LIN {X 0,Y 70.447,Z 469.266,A -85,B 0,C 180,E1 -28680.082,E2 -28680.082} C_VEL
LIN {X 0,Y 65.543,Z 474.999,A -85,B 0,C 180,E1 -28687.961,E2 -28687.961} C_VEL
LIN {X 0,Y 61.67,Z 479.556,A -85,B 0,C 180,E1 -28696.828,E2 -28696.828} C_VEL
LIN {X 0,Y 59.842,Z 481.977,A -85,B 0,C 180,E1 -28703.259,E2 -28703.259} C_VEL
LIN {X 0,Y 58.773,Z 483.966,A -85,B 0,C 180,E1 -28710.003,E2 -28710.003} C_VEL
LIN {X 0,Y 58.612,Z 485.529,A -85,B 0,C 180,E1 -28716.889,E2 -28716.889} C_VEL
LIN {X 0,Y 59.031,Z 486.685,A -85,B 0,C 180,E1 -28723.778,E2 -28723.778} C_VEL
LIN {X 0,Y 62.036,Z 487.812,A -85,B 0,C 180,E1 -28736.949,E2 -28736.949} C_VEL
LIN {X 0,Y 64.57,Z 487.807,A -85,B 0,C 180,E1 -28742.974,E2 -28742.974} C_VEL
LIN {X 0,Y 67.683,Z 487.381,A -85,B 0,C 180,E1 -28748.539,E2 -28748.539} C_VEL
LIN {X 0,Y 75.513,Z 485.311,A -85,B 0,C 180,E1 -28758.123,E2 -28758.123} C_VEL
LIN {X 0,Y 82.416,Z 482.653,A -85,B 0,C 180,E1 -28764.108,E2 -28764.108} C_VEL
LIN {X 0,Y 90.002,Z 478.961,A -85,B 0,C 180,E1 -28769.201,E2 -28769.201} C_VEL
LIN {X 0,Y 98.155,Z 474.117,A -85,B 0,C 180,E1 -28773.512,E2 -28773.512} C_VEL
LIN {X 0,Y 106.718,Z 467.974,A -85,B 0,C 180,E1 -28777.218,E2 -28777.218} C_VEL
LIN {X 0,Y 115.661,Z 460.196,A -85,B 0,C 180,E1 -28780.364,E2 -28780.364} C_VEL
LIN {X 0,Y 123.256,Z 452.216,A -85,B 0,C 180,E1 -28782.761,E2 -28782.761} C_VEL
LIN {X 0,Y 131.028,Z 442.412,A -85,B 0,C 180,E1 -28784.901,E2 -28784.901} C_VEL
LIN {X 0,Y 137.326,Z 432.712,A -85,B 0,C 180,E1 -28786.501,E2 -28786.501} C_VEL
LIN {X 0,Y 142.896,Z 422.116,A -85,B 0,C 180,E1 -28787.824,E2 -28787.824} C_VEL
LIN {X 0,Y 147.891,Z 409.841,A -85,B 0,C 180,E1 -28788.973,E2 -28788.973} C_VEL
LIN {X 0,Y 151.141,Z 398.97,A -85,B 0,C 180,E1 -28789.804,E2 -28789.804} C_VEL
LIN {X 0,Y 150.531,Z 395.282,A -85,B 0,C 180,E1 -28792.96,E2 -28792.96} C_VEL
LIN {X 0,Y 149.955,Z 392.561,A -85,B 0,C 180,E1 -28796.305,E2 -28796.305} C_VEL
LIN {X 0,Y 149.616,Z 389.913,A -85,B 0,C 180,E1 -28800.601,E2 -28800.601} C_VEL
LIN {X 0,Y 149.627,Z 390.098,A -85,B 0,C 180,E1 -28805.39,E2 -28805.39} C_VEL
LIN {X 0,Y 150.016,Z 392.663,A -85,B 0,C 180,E1 -28809.386,E2 -28809.386} C_VEL
LIN {X 0,Y 150.407,Z 397.16,A -85,B 0,C 180,E1 -28812.671,E2 -28812.671} C_VEL
LIN {X 0,Y 150.734,Z 401.874,A -85,B 0,C 180,E1 -28815.292,E2 -28815.292} C_VEL
LIN {X 0,Y 150.821,Z 403.374,A -85,B 0,C 180,E1 -28816.026,E2 -28816.026} C_VEL
LIN {X 0,Y 147.223,Z 416.009,A -85,B 0,C 180,E1 -28816.575,E2 -28816.575} C_VEL
LIN {X 0,Y 142.068,Z 428.741,A -85,B 0,C 180,E1 -28817.298,E2 -28817.298} C_VEL
LIN {X 0,Y 136.738,Z 439.083,A -85,B 0,C 180,E1 -28818.15,E2 -28818.15} C_VEL
LIN {X 0,Y 129.462,Z 450.457,A -85,B 0,C 180,E1 -28819.399,E2 -28819.399} C_VEL
LIN {X 0,Y 122.131,Z 459.743,A -85,B 0,C 180,E1 -28820.754,E2 -28820.754} C_VEL
LIN {X 0,Y 114.125,Z 468.25,A -85,B 0,C 180,E1 -28822.522,E2 -28822.522} C_VEL
LIN {X 0,Y 104.793,Z 476.609,A -85,B 0,C 180,E1 -28825.124,E2 -28825.124} C_VEL
LIN {X 0,Y 95.791,Z 483.396,A -85,B 0,C 180,E1 -28828.306,E2 -28828.306} C_VEL
LIN {X 0,Y 87.25,Z 488.876,A -85,B 0,C 180,E1 -28832.243,E2 -28832.243} C_VEL
LIN {X 0,Y 79.297,Z 493.214,A -85,B 0,C 180,E1 -28837.091,E2 -28837.091} C_VEL
LIN {X 0,Y 72.131,Z 496.518,A -85,B 0,C 180,E1 -28843.002,E2 -28843.002} C_VEL
LIN {X 0,Y 66.035,Z 498.921,A -85,B 0,C 180,E1 -28850.312,E2 -28850.312} C_VEL
LIN {X 0,Y 60.021,Z 500.751,A -85,B 0,C 180,E1 -28862.069,E2 -28862.069} C_VEL
LIN {X 0,Y 57.294,Z 501.014,A -85,B 0,C 180,E1 -28875.796,E2 -28875.796} C_VEL
LIN {X 0,Y 57.248,Z 500.581,A -85,B 0,C 180,E1 -28882.946,E2 -28882.946} C_VEL
LIN {X 0,Y 57.565,Z 499.702,A -85,B 0,C 180,E1 -28889.997,E2 -28889.997} C_VEL
LIN {X 0,Y 56.925,Z 497.644,A -85,B 0,C 180,E1 -28899.01,E2 -28899.01} C_VEL
LIN {X 0,Y 58.021,Z 493.667,A -85,B 0,C 180,E1 -28911.305,E2 -28911.305} C_VEL
LIN {X 0,Y 61.036,Z 489.039,A -85,B 0,C 180,E1 -28921.204,E2 -28921.204} C_VEL
LIN {X 0,Y 65.752,Z 483.202,A -85,B 0,C 180,E1 -28929.886,E2 -28929.886} C_VEL
LIN {X 0,Y 71.676,Z 476.201,A -85,B 0,C 180,E1 -28936.923,E2 -28936.923} C_VEL
LIN {X 0,Y 77.718,Z 468.516,A -85,B 0,C 180,E1 -28942.298,E2 -28942.298} C_VEL
LIN {X 0,Y 84.172,Z 459.58,A -85,B 0,C 180,E1 -28946.606,E2 -28946.606} C_VEL
LIN {X 0,Y 90.425,Z 449.814,A -85,B 0,C 180,E1 -28949.837,E2 -28949.837} C_VEL
LIN {X 0,Y 96.198,Z 439.132,A -85,B 0,C 180,E1 -28952.347,E2 -28952.347} C_VEL
LIN {X 0,Y 101.393,Z 427.216,A -85,B 0,C 180,E1 -28954.294,E2 -28954.294} C_VEL
LIN {X 0,Y 105.04,Z 416.019,A -85,B 0,C 180,E1 -28955.723,E2 -28955.723} C_VEL
LIN {X 0,Y 108.241,Z 402.728,A -85,B 0,C 180,E1 -28956.821,E2 -28956.821} C_VEL
LIN {X 0,Y 109.772,Z 392.127,A -85,B 0,C 180,E1 -28957.466,E2 -28957.466} C_VEL
LIN {X 0,Y 110.973,Z 365.531,A -85,B 0,C 180,E1 -28960.114,E2 -28960.114} C_VEL
LIN {X 0,Y 109.223,Z 357.79,A -85,B 0,C 180,E1 -28963.53,E2 -28963.53} C_VEL
LIN {X 0,Y 108.11,Z 353.863,A -85,B 0,C 180,E1 -28965.872,E2 -28965.872} C_VEL
LIN {X 0,Y 105.989,Z 349.494,A -85,B 0,C 180,E1 -28970.699,E2 -28970.699} C_VEL
LIN {X 0,Y 104.42,Z 345.907,A -85,B 0,C 180,E1 -28976.142,E2 -28976.142} C_VEL
LIN {X 0,Y 103.537,Z 344.387,A -85,B 0,C 180,E1 -28981.946,E2 -28981.946} C_VEL
LIN {X 0,Y 103.451,Z 344.664,A -85,B 0,C 180,E1 -28987.191,E2 -28987.191} C_VEL
LIN {X 0,Y 104.475,Z 346.425,A -85,B 0,C 180,E1 -28994.064,E2 -28994.064} C_VEL
LIN {X 0,Y 106.553,Z 350.841,A -85,B 0,C 180,E1 -29000.594,E2 -29000.594} C_VEL
LIN {X 0,Y 108.008,Z 353.756,A -85,B 0,C 180,E1 -29003.754,E2 -29003.754} C_VEL
LIN {X 0,Y 108.709,Z 356.397,A -85,B 0,C 180,E1 -29005.311,E2 -29005.311} C_VEL
LIN {X 0,Y 109.207,Z 360.955,A -85,B 0,C 180,E1 -29006.812,E2 -29006.812} C_VEL
LIN {X 0,Y 109.23,Z 367.561,A -85,B 0,C 180,E1 -29007.963,E2 -29007.963} C_VEL
LIN {X 0,Y 108.881,Z 373.098,A -85,B 0,C 180,E1 -29008.445,E2 -29008.445} C_VEL
LIN {X 0,Y 107.012,Z 388.802,A -85,B 0,C 180,E1 -29009.289,E2 -29009.289} C_VEL
LIN {X 0,Y 104.517,Z 401.209,A -85,B 0,C 180,E1 -29010.506,E2 -29010.506} C_VEL
LIN {X 0,Y 100.523,Z 414.13,A -85,B 0,C 180,E1 -29012.177,E2 -29012.177} C_VEL
LIN {X 0,Y 95.684,Z 425.905,A -85,B 0,C 180,E1 -29014.283,E2 -29014.283} C_VEL
LIN {X 0,Y 90.161,Z 436.672,A -85,B 0,C 180,E1 -29016.972,E2 -29016.972} C_VEL
LIN {X 0,Y 83.395,Z 447.397,A -85,B 0,C 180,E1 -29020.676,E2 -29020.676} C_VEL
LIN {X 0,Y 76.964,Z 456.117,A -85,B 0,C 180,E1 -29024.957,E2 -29024.957} C_VEL
LIN {X 0,Y 70.909,Z 463.33,A -85,B 0,C 180,E1 -29029.896,E2 -29029.896} C_VEL
LIN {X 0,Y 64.431,Z 470.429,A -85,B 0,C 180,E1 -29036.952,E2 -29036.952} C_VEL
LIN {X 0,Y 59.068,Z 476.085,A -85,B 0,C 180,E1 -29045.394,E2 -29045.394} C_VEL
LIN {X 0,Y 54.818,Z 480.587,A -85,B 0,C 180,E1 -29055.146,E2 -29055.146} C_VEL
LIN {X 0,Y 52.812,Z 482.982,A -85,B 0,C 180,E1 -29062.356,E2 -29062.356} C_VEL
LIN {X 0,Y 51.698,Z 484.945,A -85,B 0,C 180,E1 -29070.003,E2 -29070.003} C_VEL
LIN {X 0,Y 51.576,Z 486.482,A -85,B 0,C 180,E1 -29077.835,E2 -29077.835} C_VEL
LIN {X 0,Y 53.589,Z 488.324,A -85,B 0,C 180,E1 -29093.171,E2 -29093.171} C_VEL
LIN {X 0,Y 58.717,Z 488.646,A -85,B 0,C 180,E1 -29106.762,E2 -29106.762} C_VEL
LIN {X 0,Y 66.35,Z 487.325,A -85,B 0,C 180,E1 -29117.858,E2 -29117.858} C_VEL
LIN {X 0,Y 74.884,Z 484.742,A -85,B 0,C 180,E1 -29125.727,E2 -29125.727} C_VEL
LIN {X 0,Y 83.797,Z 481,A -85,B 0,C 180,E1 -29131.72,E2 -29131.72} C_VEL
LIN {X 0,Y 92.263,Z 476.49,A -85,B 0,C 180,E1 -29136.078,E2 -29136.078} C_VEL
LIN {X 0,Y 101.725,Z 470.278,A -85,B 0,C 180,E1 -29139.966,E2 -29139.966} C_VEL
LIN {X 0,Y 110.327,Z 463.441,A -85,B 0,C 180,E1 -29142.848,E2 -29142.848} C_VEL
LIN {X 0,Y 118.172,Z 455.983,A -85,B 0,C 180,E1 -29145.112,E2 -29145.112} C_VEL
LIN {X 0,Y 125.546,Z 447.599,A -85,B 0,C 180,E1 -29147.06,E2 -29147.06} C_VEL
LIN {X 0,Y 132.576,Z 437.981,A -85,B 0,C 180,E1 -29148.727,E2 -29148.727} C_VEL
LIN {X 0,Y 139.093,Z 426.891,A -85,B 0,C 180,E1 -29150.158,E2 -29150.158} C_VEL
LIN {X 0,Y 144.276,Z 415.747,A -85,B 0,C 180,E1 -29151.226,E2 -29151.226} C_VEL
LIN {X 0,Y 148.596,Z 403.386,A -85,B 0,C 180,E1 -29152.184,E2 -29152.184} C_VEL
LIN {X 0,Y 148.295,Z 400.667,A -85,B 0,C 180,E1 -29155.072,E2 -29155.072} C_VEL
LIN {X 0,Y 148.164,Z 399.039,A -85,B 0,C 180,E1 -29157.281,E2 -29157.281} C_VEL
LIN {X 0,Y 148.136,Z 396.81,A -85,B 0,C 180,E1 -29161.215,E2 -29161.215} C_VEL
LIN {X 0,Y 148.216,Z 397.255,A -85,B 0,C 180,E1 -29165.441,E2 -29165.441} C_VEL
LIN {X 0,Y 148.374,Z 399.308,A -85,B 0,C 180,E1 -29168.529,E2 -29168.529} C_VEL
LIN {X 0,Y 148.457,Z 403.426,A -85,B 0,C 180,E1 -29171.607,E2 -29171.607} C_VEL
LIN {X 0,Y 148.414,Z 406.748,A -85,B 0,C 180,E1 -29173.508,E2 -29173.508} C_VEL
LIN {X 0,Y 144.371,Z 419.061,A -85,B 0,C 180,E1 -29173.998,E2 -29173.998} C_VEL
LIN {X 0,Y 138.867,Z 431.453,A -85,B 0,C 180,E1 -29174.699,E2 -29174.699} C_VEL
LIN {X 0,Y 132.557,Z 442.5,A -85,B 0,C 180,E1 -29175.58,E2 -29175.58} C_VEL
LIN {X 0,Y 124.784,Z 453.466,A -85,B 0,C 180,E1 -29176.772,E2 -29176.772} C_VEL
LIN {X 0,Y 116.503,Z 462.967,A -85,B 0,C 180,E1 -29178.173,E2 -29178.173} C_VEL
LIN {X 0,Y 106.777,Z 472.17,A -85,B 0,C 180,E1 -29180.292,E2 -29180.292} C_VEL
LIN {X 0,Y 97.276,Z 479.636,A -85,B 0,C 180,E1 -29182.902,E2 -29182.902} C_VEL
LIN {X 0,Y 89.595,Z 484.749,A -85,B 0,C 180,E1 -29185.566,E2 -29185.566} C_VEL
LIN {X 0,Y 80.779,Z 489.774,A -85,B 0,C 180,E1 -29189.537,E2 -29189.537} C_VEL
LIN {X 0,Y 72.531,Z 493.714,A -85,B 0,C 180,E1 -29194.549,E2 -29194.549} C_VEL
LIN {X 0,Y 65.066,Z 496.673,A -85,B 0,C 180,E1 -29200.877,E2 -29200.877} C_VEL
LIN {X 0,Y 56.872,Z 499.214,A -85,B 0,C 180,E1 -29211.836,E2 -29211.836} C_VEL
LIN {X 0,Y 53.821,Z 499.912,A -85,B 0,C 180,E1 -29218.509,E2 -29218.509} C_VEL
LIN {X 0,Y 50.401,Z 500.122,A -85,B 0,C 180,E1 -29233.803,E2 -29233.803} C_VEL
LIN {X 0,Y 50.186,Z 499.67,A -85,B 0,C 180,E1 -29241.947,E2 -29241.947} C_VEL
LIN {X 0,Y 50.425,Z 498.764,A -85,B 0,C 180,E1 -29249.997,E2 -29249.997} C_VEL
LIN {X 0,Y 49.869,Z 496.863,A -85,B 0,C 180,E1 -29259.43,E2 -29259.43} C_VEL
LIN {X 0,Y 51.386,Z 492.633,A -85,B 0,C 180,E1 -29274.22,E2 -29274.22} C_VEL
LIN {X 0,Y 55.007,Z 487.953,A -85,B 0,C 180,E1 -29285.091,E2 -29285.091} C_VEL
LIN {X 0,Y 61.461,Z 480.978,A -85,B 0,C 180,E1 -29295.489,E2 -29295.489} C_VEL
LIN {X 0,Y 68.354,Z 473.455,A -85,B 0,C 180,E1 -29302.58,E2 -29302.58} C_VEL
LIN {X 0,Y 74.892,Z 465.553,A -85,B 0,C 180,E1 -29307.62,E2 -29307.62} C_VEL
LIN {X 0,Y 81.95,Z 456.217,A -85,B 0,C 180,E1 -29311.519,E2 -29311.519} C_VEL
LIN {X 0,Y 88.517,Z 445.782,A -85,B 0,C 180,E1 -29314.567,E2 -29314.567} C_VEL
LIN {X 0,Y 93.844,Z 435.85,A -85,B 0,C 180,E1 -29316.542,E2 -29316.542} C_VEL
LIN {X 0,Y 98.476,Z 425.238,A -85,B 0,C 180,E1 -29318.083,E2 -29318.083} C_VEL
LIN {X 0,Y 102.478,Z 413.06,A -85,B 0,C 180,E1 -29319.462,E2 -29319.462} C_VEL
LIN {X 0,Y 105.55,Z 400.127,A -85,B 0,C 180,E1 -29320.359,E2 -29320.359} C_VEL
LIN {X 0,Y 106.729,Z 391.231,A -85,B 0,C 180,E1 -29320.965,E2 -29320.965} C_VEL
LIN {X 0,Y 108.024,Z 368.585,A -85,B 0,C 180,E1 -29323.22,E2 -29323.22} C_VEL
LIN {X 0,Y 106.621,Z 361.484,A -85,B 0,C 180,E1 -29326.662,E2 -29326.662} C_VEL
LIN {X 0,Y 105.979,Z 359.172,A -85,B 0,C 180,E1 -29328.283,E2 -29328.283} C_VEL
LIN {X 0,Y 104.416,Z 355.746,A -85,B 0,C 180,E1 -29332.508,E2 -29332.508} C_VEL
LIN {X 0,Y 103.344,Z 352.817,A -85,B 0,C 180,E1 -29336.954,E2 -29336.954} C_VEL
LIN {X 0,Y 102.661,Z 351.475,A -85,B 0,C 180,E1 -29341.962,E2 -29341.962} C_VEL
LIN {X 0,Y 102.549,Z 351.619,A -85,B 0,C 180,E1 -29346.442,E2 -29346.442} C_VEL
LIN {X 0,Y 103.37,Z 353.327,A -85,B 0,C 180,E1 -29353.18,E2 -29353.18} C_VEL
LIN {X 0,Y 105.031,Z 357.268,A -85,B 0,C 180,E1 -29359.166,E2 -29359.166} C_VEL
LIN {X 0,Y 106.575,Z 360.803,A -85,B 0,C 180,E1 -29362.922,E2 -29362.922} C_VEL
LIN {X 0,Y 108.536,Z 365.675,A -85,B 0,C 180,E1 -29366.754,E2 -29366.754} C_VEL
LIN {X 0,Y 109.316,Z 367.857,A -85,B 0,C 180,E1 -29368.117,E2 -29368.117} C_VEL
LIN {X 0,Y 108.881,Z 373.098,A -85,B 0,C 180,E1 -29368.445,E2 -29368.445} C_VEL
LIN {X 0,Y 108.253,Z 377.039,A -85,B 0,C 180,E1 -29368.32,E2 -29368.32} C_VEL
LIN {X 0,Y 104.509,Z 389.408,A -85,B 0,C 180,E1 -29366.128,E2 -29366.128} C_VEL
LIN {X 0,Y 103.578,Z 393.271,A -85,B 0,C 180,E1 -29366.118,E2 -29366.118} C_VEL
LIN {X 0,Y 100.235,Z 406.705,A -85,B 0,C 180,E1 -29367.433,E2 -29367.433} C_VEL
LIN {X 0,Y 96.356,Z 417.755,A -85,B 0,C 180,E1 -29368.931,E2 -29368.931} C_VEL
LIN {X 0,Y 91.21,Z 429.048,A -85,B 0,C 180,E1 -29371,E2 -29371} C_VEL
LIN {X 0,Y 84.698,Z 440.498,A -85,B 0,C 180,E1 -29373.93,E2 -29373.93} C_VEL
LIN {X 0,Y 77.607,Z 450.682,A -85,B 0,C 180,E1 -29377.596,E2 -29377.596} C_VEL
LIN {X 0,Y 70.854,Z 458.947,A -85,B 0,C 180,E1 -29381.938,E2 -29381.938} C_VEL
LIN {X 0,Y 63.251,Z 467.05,A -85,B 0,C 180,E1 -29388.193,E2 -29388.193} C_VEL
LIN {X 0,Y 56.537,Z 473.571,A -85,B 0,C 180,E1 -29395.991,E2 -29395.991} C_VEL
LIN {X 0,Y 51.006,Z 478.774,A -85,B 0,C 180,E1 -29405.588,E2 -29405.588} C_VEL
LIN {X 0,Y 46.835,Z 482.865,A -85,B 0,C 180,E1 -29416.996,E2 -29416.996} C_VEL
LIN {X 0,Y 44.622,Z 485.924,A -85,B 0,C 180,E1 -29430.004,E2 -29430.004} C_VEL
LIN {X 0,Y 44.545,Z 487.425,A -85,B 0,C 180,E1 -29439.081,E2 -29439.081} C_VEL
LIN {X 0,Y 47.108,Z 489.218,A -85,B 0,C 180,E1 -29456.591,E2 -29456.591} C_VEL
LIN {X 0,Y 49.75,Z 489.55,A -85,B 0,C 180,E1 -29464.41,E2 -29464.41} C_VEL
LIN {X 0,Y 53.173,Z 489.475,A -85,B 0,C 180,E1 -29471.369,E2 -29471.369} C_VEL
LIN {X 0,Y 61.785,Z 488.103,A -85,B 0,C 180,E1 -29482.776,E2 -29482.776} C_VEL
LIN {X 0,Y 70.595,Z 485.633,A -85,B 0,C 180,E1 -29490.146,E2 -29490.146} C_VEL
LIN {X 0,Y 80.655,Z 481.654,A -85,B 0,C 180,E1 -29496.199,E2 -29496.199} C_VEL
LIN {X 0,Y 89.599,Z 477.09,A -85,B 0,C 180,E1 -29500.266,E2 -29500.266} C_VEL
LIN {X 0,Y 99.26,Z 470.984,A -85,B 0,C 180,E1 -29503.768,E2 -29503.768} C_VEL
LIN {X 0,Y 108.438,Z 463.909,A -85,B 0,C 180,E1 -29506.451,E2 -29506.451} C_VEL
LIN {X 0,Y 116.537,Z 456.373,A -85,B 0,C 180,E1 -29508.52,E2 -29508.52} C_VEL
LIN {X 0,Y 124.823,Z 447.046,A -85,B 0,C 180,E1 -29510.431,E2 -29510.431} C_VEL
LIN {X 0,Y 132.197,Z 436.814,A -85,B 0,C 180,E1 -29511.956,E2 -29511.956} C_VEL
LIN {X 0,Y 138.886,Z 425.243,A -85,B 0,C 180,E1 -29513.253,E2 -29513.253} C_VEL
LIN {X 0,Y 144.399,Z 412.783,A -85,B 0,C 180,E1 -29514.26,E2 -29514.26} C_VEL
LIN {X 0,Y 145.466,Z 409.899,A -85,B 0,C 180,E1 -29514.454,E2 -29514.454} C_VEL
LIN {X 0,Y 146.057,Z 407.902,A -85,B 0,C 180,E1 -29514.864,E2 -29514.864} C_VEL
LIN {X 0,Y 146.1,Z 405.985,A -85,B 0,C 180,E1 -29517.242,E2 -29517.242} C_VEL
LIN {X 0,Y 146.312,Z 403.721,A -85,B 0,C 180,E1 -29521.23,E2 -29521.23} C_VEL
LIN {X 0,Y 146.408,Z 404.029,A -85,B 0,C 180,E1 -29524.991,E2 -29524.991} C_VEL
LIN {X 0,Y 146.409,Z 405.827,A -85,B 0,C 180,E1 -29527.672,E2 -29527.672} C_VEL
LIN {X 0,Y 146.272,Z 408.355,A -85,B 0,C 180,E1 -29529.682,E2 -29529.682} C_VEL
LIN {X 0,Y 146.187,Z 409.407,A -85,B 0,C 180,E1 -29530.387,E2 -29530.387} C_VEL
LIN {X 0,Y 145.896,Z 410.931,A -85,B 0,C 180,E1 -29530.954,E2 -29530.954} C_VEL
LIN {X 0,Y 141.073,Z 423.557,A -85,B 0,C 180,E1 -29531.415,E2 -29531.415} C_VEL
LIN {X 0,Y 135.618,Z 434.514,A -85,B 0,C 180,E1 -29532.025,E2 -29532.025} C_VEL
LIN {X 0,Y 128.848,Z 445.335,A -85,B 0,C 180,E1 -29532.841,E2 -29532.841} C_VEL
LIN {X 0,Y 121.234,Z 455.208,A -85,B 0,C 180,E1 -29533.831,E2 -29533.831} C_VEL
LIN {X 0,Y 112.813,Z 464.214,A -85,B 0,C 180,E1 -29535.068,E2 -29535.068} C_VEL
LIN {X 0,Y 102.875,Z 473.063,A -85,B 0,C 180,E1 -29536.975,E2 -29536.975} C_VEL
LIN {X 0,Y 93.121,Z 480.178,A -85,B 0,C 180,E1 -29539.369,E2 -29539.369} C_VEL
LIN {X 0,Y 83.635,Z 485.935,A -85,B 0,C 180,E1 -29542.428,E2 -29542.428} C_VEL
LIN {X 0,Y 74.53,Z 490.533,A -85,B 0,C 180,E1 -29546.382,E2 -29546.382} C_VEL
LIN {X 0,Y 65.954,Z 494.092,A -85,B 0,C 180,E1 -29551.515,E2 -29551.515} C_VEL
LIN {X 0,Y 60.627,Z 495.913,A -85,B 0,C 180,E1 -29555.759,E2 -29555.759} C_VEL
LIN {X 0,Y 51.451,Z 498.411,A -85,B 0,C 180,E1 -29566.92,E2 -29566.92} C_VEL
LIN {X 0,Y 45.181,Z 499.328,A -85,B 0,C 180,E1 -29582.179,E2 -29582.179} C_VEL
LIN {X 0,Y 43.151,Z 498.759,A -85,B 0,C 180,E1 -29600.623,E2 -29600.623} C_VEL
LIN {X 0,Y 43.281,Z 497.814,A -85,B 0,C 180,E1 -29609.996,E2 -29609.996} C_VEL
LIN {X 0,Y 42.808,Z 496.092,A -85,B 0,C 180,E1 -29619.927,E2 -29619.927} C_VEL
LIN {X 0,Y 44.937,Z 491.595,A -85,B 0,C 180,E1 -29637.977,E2 -29637.977} C_VEL
LIN {X 0,Y 49.305,Z 486.857,A -85,B 0,C 180,E1 -29649.893,E2 -29649.893} C_VEL
LIN {X 0,Y 55.556,Z 480.89,A -85,B 0,C 180,E1 -29659.372,E2 -29659.372} C_VEL
LIN {X 0,Y 63.052,Z 473.46,A -85,B 0,C 180,E1 -29666.711,E2 -29666.711} C_VEL
LIN {X 0,Y 71.308,Z 464.232,A -85,B 0,C 180,E1 -29672.494,E2 -29672.494} C_VEL
LIN {X 0,Y 78.769,Z 454.749,A -85,B 0,C 180,E1 -29676.131,E2 -29676.131} C_VEL
LIN {X 0,Y 85.705,Z 444.204,A -85,B 0,C 180,E1 -29678.862,E2 -29678.862} C_VEL
LIN {X 0,Y 92.059,Z 432.522,A -85,B 0,C 180,E1 -29680.854,E2 -29680.854} C_VEL
LIN {X 0,Y 96.682,Z 421.55,A -85,B 0,C 180,E1 -29682.267,E2 -29682.267} C_VEL
LIN {X 0,Y 100.751,Z 408.535,A -85,B 0,C 180,E1 -29683.46,E2 -29683.46} C_VEL
LIN {X 0,Y 103.545,Z 395.546,A -85,B 0,C 180,E1 -29684.178,E2 -29684.178} C_VEL
LIN {X 0,Y 105.35,Z 372.33,A -85,B 0,C 180,E1 -29686.437,E2 -29686.437} C_VEL
LIN {X 0,Y 105.326,Z 371.094,A -85,B 0,C 180,E1 -29686.741,E2 -29686.741} C_VEL
LIN {X 0,Y 104.413,Z 365.618,A -85,B 0,C 180,E1 -29689.701,E2 -29689.701} C_VEL
LIN {X 0,Y 103.08,Z 362.271,A -85,B 0,C 180,E1 -29693.885,E2 -29693.885} C_VEL
LIN {X 0,Y 102.244,Z 359.665,A -85,B 0,C 180,E1 -29698.031,E2 -29698.031} C_VEL
LIN {X 0,Y 101.779,Z 358.611,A -85,B 0,C 180,E1 -29701.979,E2 -29701.979} C_VEL
LIN {X 0,Y 101.662,Z 358.524,A -85,B 0,C 180,E1 -29705.052,E2 -29705.052} C_VEL
LIN {X 0,Y 102.283,Z 360.165,A -85,B 0,C 180,E1 -29712.209,E2 -29712.209} C_VEL
LIN {X 0,Y 103.673,Z 363.973,A -85,B 0,C 180,E1 -29718.017,E2 -29718.017} C_VEL
LIN {X 0,Y 105.163,Z 367.769,A -85,B 0,C 180,E1 -29722.044,E2 -29722.044} C_VEL
LIN {X 0,Y 106.381,Z 371.345,A -85,B 0,C 180,E1 -29724.778,E2 -29724.778} C_VEL
LIN {X 0,Y 104.414,Z 388.414,A -85,B 0,C 180,E1 -29725.704,E2 -29725.704} C_VEL
LIN {X 0,Y 103.578,Z 393.271,A -85,B 0,C 180,E1 -29726.118,E2 -29726.118} C_VEL
LIN {X 0,Y 102.686,Z 397.165,A -85,B 0,C 180,E1 -29726.324,E2 -29726.324} C_VEL
LIN {X 0,Y 100.116,Z 404.548,A -85,B 0,C 180,E1 -29726.011,E2 -29726.011} C_VEL
LIN {X 0,Y 94.376,Z 417.212,A -85,B 0,C 180,E1 -29725.212,E2 -29725.212} C_VEL
LIN {X 0,Y 91.903,Z 422.493,A -85,B 0,C 180,E1 -29725.606,E2 -29725.606} C_VEL
LIN {X 0,Y 86.292,Z 433.487,A -85,B 0,C 180,E1 -29727.669,E2 -29727.669} C_VEL
LIN {X 0,Y 79.488,Z 444.166,A -85,B 0,C 180,E1 -29730.458,E2 -29730.458} C_VEL
LIN {X 0,Y 72.07,Z 453.796,A -85,B 0,C 180,E1 -29734.021,E2 -29734.021} C_VEL
LIN {X 0,Y 64.976,Z 461.682,A -85,B 0,C 180,E1 -29738.361,E2 -29738.361} C_VEL
LIN {X 0,Y 56.929,Z 469.437,A -85,B 0,C 180,E1 -29744.783,E2 -29744.783} C_VEL
LIN {X 0,Y 50.858,Z 474.704,A -85,B 0,C 180,E1 -29751.554,E2 -29751.554} C_VEL
LIN {X 0,Y 44.685,Z 479.848,A -85,B 0,C 180,E1 -29761.852,E2 -29761.852} C_VEL
LIN {X 0,Y 39.951,Z 483.895,A -85,B 0,C 180,E1 -29774.705,E2 -29774.705} C_VEL
LIN {X 0,Y 37.542,Z 486.904,A -85,B 0,C 180,E1 -29790.004,E2 -29790.004} C_VEL
LIN {X 0,Y 37.546,Z 488.36,A -85,B 0,C 180,E1 -29800.793,E2 -29800.793} C_VEL
LIN {X 0,Y 40.866,Z 490.109,A -85,B 0,C 180,E1 -29821.064,E2 -29821.064} C_VEL
LIN {X 0,Y 44.047,Z 490.419,A -85,B 0,C 180,E1 -29829.663,E2 -29829.663} C_VEL
LIN {X 0,Y 48.042,Z 490.3,A -85,B 0,C 180,E1 -29837.011,E2 -29837.011} C_VEL
LIN {X 0,Y 57.745,Z 488.881,A -85,B 0,C 180,E1 -29848.428,E2 -29848.428} C_VEL
LIN {X 0,Y 66.842,Z 486.506,A -85,B 0,C 180,E1 -29855.127,E2 -29855.127} C_VEL
LIN {X 0,Y 74.98,Z 483.588,A -85,B 0,C 180,E1 -29859.609,E2 -29859.609} C_VEL
LIN {X 0,Y 84.277,Z 479.361,A -85,B 0,C 180,E1 -29863.54,E2 -29863.54} C_VEL
LIN {X 0,Y 93.873,Z 473.916,A -85,B 0,C 180,E1 -29866.725,E2 -29866.725} C_VEL
LIN {X 0,Y 103.672,Z 467.058,A -85,B 0,C 180,E1 -29869.41,E2 -29869.41} C_VEL
LIN {X 0,Y 113.65,Z 458.379,A -85,B 0,C 180,E1 -29871.661,E2 -29871.661} C_VEL
LIN {X 0,Y 122.172,Z 449.293,A -85,B 0,C 180,E1 -29873.393,E2 -29873.393} C_VEL
LIN {X 0,Y 129.68,Z 439.505,A -85,B 0,C 180,E1 -29874.767,E2 -29874.767} C_VEL
LIN {X 0,Y 136.426,Z 428.519,A -85,B 0,C 180,E1 -29875.914,E2 -29875.914} C_VEL
LIN {X 0,Y 142.125,Z 416.7,A -85,B 0,C 180,E1 -29876.833,E2 -29876.833} C_VEL
LIN {X 0,Y 143.174,Z 414.132,A -85,B 0,C 180,E1 -29877.001,E2 -29877.001} C_VEL
LIN {X 0,Y 143.579,Z 413,A -85,B 0,C 180,E1 -29877.194,E2 -29877.194} C_VEL
LIN {X 0,Y 143.873,Z 411.351,A -85,B 0,C 180,E1 -29879.999,E2 -29879.999} C_VEL
LIN {X 0,Y 144.164,Z 410.453,A -85,B 0,C 180,E1 -29882.794,E2 -29882.794} C_VEL
LIN {X 0,Y 144.189,Z 411.309,A -85,B 0,C 180,E1 -29885.594,E2 -29885.594} C_VEL
LIN {X 0,Y 143.914,Z 413.75,A -85,B 0,C 180,E1 -29888.106,E2 -29888.106} C_VEL
LIN {X 0,Y 143.036,Z 416.171,A -85,B 0,C 180,E1 -29888.334,E2 -29888.334} C_VEL
LIN {X 0,Y 138.093,Z 427.417,A -85,B 0,C 180,E1 -29888.718,E2 -29888.718} C_VEL
LIN {X 0,Y 131.704,Z 438.837,A -85,B 0,C 180,E1 -29889.298,E2 -29889.298} C_VEL
LIN {X 0,Y 124.029,Z 449.72,A -85,B 0,C 180,E1 -29890.087,E2 -29890.087} C_VEL
LIN {X 0,Y 114.602,Z 460.471,A -85,B 0,C 180,E1 -29891.126,E2 -29891.126} C_VEL
LIN {X 0,Y 106.08,Z 468.429,A -85,B 0,C 180,E1 -29892.253,E2 -29892.253} C_VEL
LIN {X 0,Y 95.997,Z 476.264,A -85,B 0,C 180,E1 -29894.058,E2 -29894.058} C_VEL
LIN {X 0,Y 84.431,Z 483.538,A -85,B 0,C 180,E1 -29896.811,E2 -29896.811} C_VEL
LIN {X 0,Y 74.788,Z 488.455,A -85,B 0,C 180,E1 -29899.992,E2 -29899.992} C_VEL
LIN {X 0,Y 65.511,Z 492.294,A -85,B 0,C 180,E1 -29904.23,E2 -29904.23} C_VEL
LIN {X 0,Y 56.751,Z 495.154,A -85,B 0,C 180,E1 -29909.898,E2 -29909.898} C_VEL
LIN {X 0,Y 46.497,Z 497.601,A -85,B 0,C 180,E1 -29920.905,E2 -29920.905} C_VEL
LIN {X 0,Y 39.002,Z 498.456,A -85,B 0,C 180,E1 -29937.272,E2 -29937.272} C_VEL
LIN {X 0,Y 36.135,Z 497.845,A -85,B 0,C 180,E1 -29958.78,E2 -29958.78} C_VEL
LIN {X 0,Y 36.135,Z 496.853,A -85,B 0,C 180,E1 -29969.995,E2 -29969.995} C_VEL
LIN {X 0,Y 35.999,Z 494.226,A -85,B 0,C 180,E1 -29987.023,E2 -29987.023} C_VEL
LIN {X 0,Y 38.741,Z 490.542,A -85,B 0,C 180,E1 -30002.966,E2 -30002.966} C_VEL
LIN {X 0,Y 44.046,Z 485.746,A -85,B 0,C 180,E1 -30015.884,E2 -30015.884} C_VEL
LIN {X 0,Y 51.182,Z 479.715,A -85,B 0,C 180,E1 -30025.468,E2 -30025.468} C_VEL
LIN {X 0,Y 59.405,Z 472.211,A -85,B 0,C 180,E1 -30032.527,E2 -30032.527} C_VEL
LIN {X 0,Y 68.305,Z 462.906,A -85,B 0,C 180,E1 -30037.814,E2 -30037.814} C_VEL
LIN {X 0,Y 76.149,Z 453.283,A -85,B 0,C 180,E1 -30041.074,E2 -30041.074} C_VEL
LIN {X 0,Y 83.409,Z 442.63,A -85,B 0,C 180,E1 -30043.414,E2 -30043.414} C_VEL
LIN {X 0,Y 89.15,Z 432.373,A -85,B 0,C 180,E1 -30044.941,E2 -30044.941} C_VEL
LIN {X 0,Y 94.059,Z 421.252,A -85,B 0,C 180,E1 -30046.237,E2 -30046.237} C_VEL
LIN {X 0,Y 98.32,Z 408.307,A -85,B 0,C 180,E1 -30047.291,E2 -30047.291} C_VEL
LIN {X 0,Y 101.193,Z 395.546,A -85,B 0,C 180,E1 -30047.944,E2 -30047.944} C_VEL
LIN {X 0,Y 103.093,Z 375.05,A -85,B 0,C 180,E1 -30049.94,E2 -30049.94} C_VEL
LIN {X 0,Y 102.812,Z 372.043,A -85,B 0,C 180,E1 -30051.401,E2 -30051.401} C_VEL
LIN {X 0,Y 101.922,Z 369.065,A -85,B 0,C 180,E1 -30054.808,E2 -30054.808} C_VEL
LIN {X 0,Y 101.199,Z 366.538,A -85,B 0,C 180,E1 -30059.006,E2 -30059.006} C_VEL
LIN {X 0,Y 100.818,Z 365.464,A -85,B 0,C 180,E1 -30063.998,E2 -30063.998} C_VEL
LIN {X 0,Y 101.205,Z 366.854,A -85,B 0,C 180,E1 -30071.01,E2 -30071.01} C_VEL
LIN {X 0,Y 102.394,Z 370.72,A -85,B 0,C 180,E1 -30076.947,E2 -30076.947} C_VEL
LIN {X 0,Y 103.6,Z 374.455,A -85,B 0,C 180,E1 -30080.735,E2 -30080.735} C_VEL
LIN {X 0,Y 103.777,Z 375.027,A -85,B 0,C 180,E1 -30081.217,E2 -30081.217} C_VEL
LIN {X 0,Y 101.723,Z 391.133,A -85,B 0,C 180,E1 -30082.15,E2 -30082.15} C_VEL
LIN {X 0,Y 99.003,Z 403.096,A -85,B 0,C 180,E1 -30083.198,E2 -30083.198} C_VEL
LIN {X 0,Y 95.243,Z 414.479,A -85,B 0,C 180,E1 -30084.458,E2 -30084.458} C_VEL
LIN {X 0,Y 91.903,Z 422.493,A -85,B 0,C 180,E1 -30085.606,E2 -30085.606} C_VEL
LIN {X 0,Y 89.242,Z 427.73,A -85,B 0,C 180,E1 -30086.068,E2 -30086.068} C_VEL
LIN {X 0,Y 83.803,Z 436.037,A -85,B 0,C 180,E1 -30085.893,E2 -30085.893} C_VEL
LIN {X 0,Y 77.722,Z 443.881,A -85,B 0,C 180,E1 -30085.862,E2 -30085.862} C_VEL
LIN {X 0,Y 74.061,Z 448.389,A -85,B 0,C 180,E1 -30086.705,E2 -30086.705} C_VEL
LIN {X 0,Y 65.333,Z 458.436,A -85,B 0,C 180,E1 -30090.627,E2 -30090.627} C_VEL
LIN {X 0,Y 57.872,Z 465.686,A -85,B 0,C 180,E1 -30094.949,E2 -30094.949} C_VEL
LIN {X 0,Y 49.465,Z 472.818,A -85,B 0,C 180,E1 -30101.769,E2 -30101.769} C_VEL
LIN {X 0,Y 43.138,Z 477.626,A -85,B 0,C 180,E1 -30109.338,E2 -30109.338} C_VEL
LIN {X 0,Y 36.565,Z 482.345,A -85,B 0,C 180,E1 -30121.287,E2 -30121.287} C_VEL
LIN {X 0,Y 31.877,Z 485.995,A -85,B 0,C 180,E1 -30137.269,E2 -30137.269} C_VEL
LIN {X 0,Y 30.463,Z 487.877,A -85,B 0,C 180,E1 -30150.006,E2 -30150.006} C_VEL
LIN {X 0,Y 30.598,Z 489.295,A -85,B 0,C 180,E1 -30163.284,E2 -30163.284} C_VEL
LIN {X 0,Y 34.958,Z 491.001,A -85,B 0,C 180,E1 -30187.099,E2 -30187.099} C_VEL
LIN {X 0,Y 38.828,Z 491.278,A -85,B 0,C 180,E1 -30196.392,E2 -30196.392} C_VEL
LIN {X 0,Y 48.713,Z 490.585,A -85,B 0,C 180,E1 -30209.961,E2 -30209.961} C_VEL
LIN {X 0,Y 54.348,Z 489.66,A -85,B 0,C 180,E1 -30214.855,E2 -30214.855} C_VEL
LIN {X 0,Y 63.584,Z 487.397,A -85,B 0,C 180,E1 -30220.633,E2 -30220.633} C_VEL
LIN {X 0,Y 72.799,Z 484.269,A -85,B 0,C 180,E1 -30224.886,E2 -30224.886} C_VEL
LIN {X 0,Y 82.538,Z 479.988,A -85,B 0,C 180,E1 -30228.3,E2 -30228.3} C_VEL
LIN {X 0,Y 93.729,Z 473.707,A -85,B 0,C 180,E1 -30231.374,E2 -30231.374} C_VEL
LIN {X 0,Y 104.301,Z 466.187,A -85,B 0,C 180,E1 -30233.662,E2 -30233.662} C_VEL
LIN {X 0,Y 114.547,Z 457.135,A -85,B 0,C 180,E1 -30235.571,E2 -30235.571} C_VEL
LIN {X 0,Y 123.766,Z 446.895,A -85,B 0,C 180,E1 -30237.078,E2 -30237.078} C_VEL
LIN {X 0,Y 130.964,Z 437.035,A -85,B 0,C 180,E1 -30238.165,E2 -30238.165} C_VEL
LIN {X 0,Y 137.338,Z 426.201,A -85,B 0,C 180,E1 -30239.104,E2 -30239.104} C_VEL
LIN {X 0,Y 140.564,Z 419.477,A -85,B 0,C 180,E1 -30239.533,E2 -30239.533} C_VEL
LIN {X 0,Y 141.136,Z 418.123,A -85,B 0,C 180,E1 -30239.999,E2 -30239.999} C_VEL
LIN {X 0,Y 141.619,Z 417.141,A -85,B 0,C 180,E1 -30242.844,E2 -30242.844} C_VEL
LIN {X 0,Y 141.224,Z 418.913,A -85,B 0,C 180,E1 -30245.559,E2 -30245.559} C_VEL
LIN {X 0,Y 135.455,Z 430.792,A -85,B 0,C 180,E1 -30245.906,E2 -30245.906} C_VEL
LIN {X 0,Y 128.106,Z 442.659,A -85,B 0,C 180,E1 -30246.414,E2 -30246.414} C_VEL
LIN {X 0,Y 120.382,Z 452.62,A -85,B 0,C 180,E1 -30247.032,E2 -30247.032} C_VEL
LIN {X 0,Y 111.716,Z 461.768,A -85,B 0,C 180,E1 -30247.767,E2 -30247.767} C_VEL
LIN {X 0,Y 101.365,Z 470.73,A -85,B 0,C 180,E1 -30248.882,E2 -30248.882} C_VEL
LIN {X 0,Y 91.113,Z 477.987,A -85,B 0,C 180,E1 -30250.428,E2 -30250.428} C_VEL
LIN {X 0,Y 79.297,Z 484.667,A -85,B 0,C 180,E1 -30252.855,E2 -30252.855} C_VEL
LIN {X 0,Y 69.38,Z 489.161,A -85,B 0,C 180,E1 -30255.773,E2 -30255.773} C_VEL
LIN {X 0,Y 59.746,Z 492.623,A -85,B 0,C 180,E1 -30259.767,E2 -30259.767} C_VEL
LIN {X 0,Y 47.648,Z 495.787,A -85,B 0,C 180,E1 -30267.745,E2 -30267.745} C_VEL
LIN {X 0,Y 42.173,Z 496.78,A -85,B 0,C 180,E1 -30273.563,E2 -30273.563} C_VEL
LIN {X 0,Y 33.225,Z 497.585,A -85,B 0,C 180,E1 -30290.606,E2 -30290.606} C_VEL
LIN {X 0,Y 29.157,Z 496.923,A -85,B 0,C 180,E1 -30316.046,E2 -30316.046} C_VEL
LIN {X 0,Y 28.989,Z 495.892,A -85,B 0,C 180,E1 -30329.994,E2 -30329.994} C_VEL
LIN {X 0,Y 29.211,Z 493.212,A -85,B 0,C 180,E1 -30351.149,E2 -30351.149} C_VEL
LIN {X 0,Y 32.94,Z 489.477,A -85,B 0,C 180,E1 -30369.789,E2 -30369.789} C_VEL
LIN {X 0,Y 39.4,Z 484.631,A -85,B 0,C 180,E1 -30383.38,E2 -30383.38} C_VEL
LIN {X 0,Y 48.778,Z 477.507,A -85,B 0,C 180,E1 -30393.736,E2 -30393.736} C_VEL
LIN {X 0,Y 58.009,Z 469.566,A -85,B 0,C 180,E1 -30399.863,E2 -30399.863} C_VEL
LIN {X 0,Y 65.946,Z 461.558,A -85,B 0,C 180,E1 -30403.552,E2 -30403.552} C_VEL
LIN {X 0,Y 74.128,Z 451.812,A -85,B 0,C 180,E1 -30406.343,E2 -30406.343} C_VEL
LIN {X 0,Y 81.669,Z 441.057,A -85,B 0,C 180,E1 -30408.185,E2 -30408.185} C_VEL
LIN {X 0,Y 87.576,Z 430.637,A -85,B 0,C 180,E1 -30409.423,E2 -30409.423} C_VEL
LIN {X 0,Y 92.617,Z 419.182,A -85,B 0,C 180,E1 -30410.545,E2 -30410.545} C_VEL
LIN {X 0,Y 96.837,Z 406.299,A -85,B 0,C 180,E1 -30411.393,E2 -30411.393} C_VEL
LIN {X 0,Y 99.478,Z 394.488,A -85,B 0,C 180,E1 -30411.944,E2 -30411.944} C_VEL
LIN {X 0,Y 101.22,Z 377.875,A -85,B 0,C 180,E1 -30413.597,E2 -30413.597} C_VEL
LIN {X 0,Y 100.738,Z 375.73,A -85,B 0,C 180,E1 -30416,E2 -30416} C_VEL
LIN {X 0,Y 100.13,Z 373.26,A -85,B 0,C 180,E1 -30420.524,E2 -30420.524} C_VEL
LIN {X 0,Y 99.946,Z 372.525,A -85,B 0,C 180,E1 -30424.033,E2 -30424.033} C_VEL
LIN {X 0,Y 100.218,Z 373.897,A -85,B 0,C 180,E1 -30430.367,E2 -30430.367} C_VEL
LIN {X 0,Y 101.116,Z 377.394,A -85,B 0,C 180,E1 -30435.718,E2 -30435.718} C_VEL
LIN {X 0,Y 101.582,Z 379.078,A -85,B 0,C 180,E1 -30437.575,E2 -30437.575} C_VEL
LIN {X 0,Y 99.559,Z 393.08,A -85,B 0,C 180,E1 -30438.371,E2 -30438.371} C_VEL
LIN {X 0,Y 96.225,Z 406.178,A -85,B 0,C 180,E1 -30439.437,E2 -30439.437} C_VEL
LIN {X 0,Y 91.881,Z 418.147,A -85,B 0,C 180,E1 -30440.729,E2 -30440.729} C_VEL
LIN {X 0,Y 86.447,Z 429.535,A -85,B 0,C 180,E1 -30442.375,E2 -30442.375} C_VEL
LIN {X 0,Y 79.326,Z 441.199,A -85,B 0,C 180,E1 -30444.762,E2 -30444.762} C_VEL
LIN {X 0,Y 74.061,Z 448.389,A -85,B 0,C 180,E1 -30446.705,E2 -30446.705} C_VEL
LIN {X 0,Y 70.237,Z 452.801,A -85,B 0,C 180,E1 -30447.674,E2 -30447.674} C_VEL
LIN {X 0,Y 60.037,Z 462.234,A -85,B 0,C 180,E1 -30448.228,E2 -30448.228} C_VEL
LIN {X 0,Y 53.948,Z 467.164,A -85,B 0,C 180,E1 -30449.301,E2 -30449.301} C_VEL
LIN {X 0,Y 51.041,Z 469.447,A -85,B 0,C 180,E1 -30450.706,E2 -30450.706} C_VEL
LIN {X 0,Y 43.608,Z 474.978,A -85,B 0,C 180,E1 -30456.319,E2 -30456.319} C_VEL
LIN {X 0,Y 35.4,Z 480.402,A -85,B 0,C 180,E1 -30465.992,E2 -30465.992} C_VEL
LIN {X 0,Y 28.432,Z 484.696,A -85,B 0,C 180,E1 -30480.379,E2 -30480.379} C_VEL
LIN {X 0,Y 25.019,Z 487,A -85,B 0,C 180,E1 -30493.693,E2 -30493.693} C_VEL
LIN {X 0,Y 23.384,Z 488.839,A -85,B 0,C 180,E1 -30510.007,E2 -30510.007} C_VEL
LIN {X 0,Y 23.742,Z 490.229,A -85,B 0,C 180,E1 -30527.225,E2 -30527.225} C_VEL
LIN {X 0,Y 29.59,Z 491.893,A -85,B 0,C 180,E1 -30555.448,E2 -30555.448} C_VEL
LIN {X 0,Y 34.297,Z 492.128,A -85,B 0,C 180,E1 -30565.058,E2 -30565.058} C_VEL
LIN {X 0,Y 45.561,Z 491.386,A -85,B 0,C 180,E1 -30577.755,E2 -30577.755} C_VEL
LIN {X 0,Y 51.721,Z 490.438,A -85,B 0,C 180,E1 -30582.03,E2 -30582.03} C_VEL
LIN {X 0,Y 61.061,Z 488.265,A -85,B 0,C 180,E1 -30586.69,E2 -30586.69} C_VEL
LIN {X 0,Y 71.274,Z 484.948,A -85,B 0,C 180,E1 -30590.425,E2 -30590.425} C_VEL
LIN {X 0,Y 81.391,Z 480.615,A -85,B 0,C 180,E1 -30593.227,E2 -30593.227} C_VEL
LIN {X 0,Y 92.422,Z 474.567,A -85,B 0,C 180,E1 -30595.638,E2 -30595.638} C_VEL
LIN {X 0,Y 102.019,Z 467.996,A -85,B 0,C 180,E1 -30597.312,E2 -30597.312} C_VEL
LIN {X 0,Y 112.469,Z 459.159,A -85,B 0,C 180,E1 -30598.899,E2 -30598.899} C_VEL
LIN {X 0,Y 121.23,Z 450.016,A -85,B 0,C 180,E1 -30600.114,E2 -30600.114} C_VEL
LIN {X 0,Y 129.358,Z 439.446,A -85,B 0,C 180,E1 -30601.123,E2 -30601.123} C_VEL
LIN {X 0,Y 136.615,Z 427.588,A -85,B 0,C 180,E1 -30602,E2 -30602} C_VEL
LIN {X 0,Y 138.493,Z 423.898,A -85,B 0,C 180,E1 -30602.219,E2 -30602.219} C_VEL
LIN {X 0,Y 138.585,Z 423.765,A -85,B 0,C 180,E1 -30602.562,E2 -30602.562} C_VEL
LIN {X 0,Y 138.161,Z 424.658,A -85,B 0,C 180,E1 -30602.774,E2 -30602.774} C_VEL
LIN {X 0,Y 131.96,Z 435.793,A -85,B 0,C 180,E1 -30603.037,E2 -30603.037} C_VEL
LIN {X 0,Y 124.091,Z 447.049,A -85,B 0,C 180,E1 -30603.429,E2 -30603.429} C_VEL
LIN {X 0,Y 116.223,Z 456.159,A -85,B 0,C 180,E1 -30603.84,E2 -30603.84} C_VEL
LIN {X 0,Y 105.742,Z 466.044,A -85,B 0,C 180,E1 -30604.469,E2 -30604.469} C_VEL
LIN {X 0,Y 95.307,Z 474.034,A -85,B 0,C 180,E1 -30605.431,E2 -30605.431} C_VEL
LIN {X 0,Y 84.911,Z 480.463,A -85,B 0,C 180,E1 -30606.666,E2 -30606.666} C_VEL
LIN {X 0,Y 74.601,Z 485.649,A -85,B 0,C 180,E1 -30608.428,E2 -30608.428} C_VEL
